               FOR #li_Counter_Hor := 1 TO 3 DO
                   FOR #li_Counter_Ver := 1 TO 3 DO
                       IF ("gtyp_VGR".s_HBW_Outsource_Typ = "gtyp_HBW".Rack_Workpiece[#li_Counter_Ver, #li_Counter_Hor].s_type)
                           AND (#lldt_Outsource > "gtyp_HBW".Rack_History[#li_Counter_Ver, #li_Counter_Hor].History[3].ldt_ts)
                           AND NOT ("gtyp_HBW".Rack_History[#li_Counter_Ver, #li_Counter_Hor].History[3].ldt_ts = LDT#1970-01-01-00:00:00) THEN
                           #lldt_Outsource := "gtyp_HBW".Rack_History[#li_Counter_Ver, #li_Counter_Hor].History[3].ldt_ts;
                           #li_Counter_Act_Hor := #li_Counter_Hor;
                           #li_Counter_Act_Ver := #li_Counter_Ver;
                           #ldi_PosRack_Horizontal := "gtyp_HBW".Rack_Pos[#li_Counter_Ver, #li_Counter_Hor].di_PosRack_Horizontal;
                           #ldi_PosRack_Vertical := "gtyp_HBW".Rack_Pos[#li_Counter_Ver, #li_Counter_Hor].di_PosRack_Vertical;
                       END_IF;
                   END_FOR;
               END_FOR;

               IF (#li_Counter_Act_Hor = 4) OR (#li_Counter_Act_Ver = 4) THEN
                   #li_StepCase := 40;
               ELSE
                   #li_StepCase := 70;
               END_IF;

           70: // Position vertical/horizontal HBW
               "gtyp_HBW".Horizontal_Axis.di_Target_Position := #ldi_PosRack_Horizontal;
               "gtyp_HBW".Horizontal_Axis.x_Start_Positioning := TRUE;
               "gtyp_HBW".Vertical_Axis.di_Target_Position := #ldi_PosRack_Vertical;
               "gtyp_HBW".Vertical_Axis.x_Start_Positioning := TRUE;

               IF ("gtyp_HBW".Horizontal_Axis.di_Actual_Position <= (#ldi_PosRack_Horizontal + "gtyp_HBW".Horizontal_Axis.Config.di_Pos_Window))
                   AND ("gtyp_HBW".Horizontal_Axis.di_Actual_Position >= (#ldi_PosRack_Horizontal - "gtyp_HBW".Horizontal_Axis.Config.di_Pos_Window))
                   AND "gtyp_HBW".Horizontal_Axis.x_Position_Reached THEN
                   "gtyp_HBW".Horizontal_Axis.x_Start_Positioning := FALSE;
               END_IF;

               IF ("gtyp_HBW".Vertical_Axis.di_Actual_Position <= (#ldi_PosRack_Vertical + "gtyp_HBW".Vertical_Axis.Config.di_Pos_Window))
                   AND ("gtyp_HBW".Vertical_Axis.di_Actual_Position >= (#ldi_PosRack_Vertical - "gtyp_HBW".Vertical_Axis.Config.di_Pos_Window))
                   AND "gtyp_HBW".Vertical_Axis.x_Position_Reached THEN
                   "gtyp_HBW".Vertical_Axis.x_Start_Positioning := FALSE;
               END_IF;

               IF ("gtyp_HBW".Horizontal_Axis.di_Actual_Position <= (#ldi_PosRack_Horizontal + "gtyp_HBW".Horizontal_Axis.Config.di_Pos_Window))
                   AND ("gtyp_HBW".Horizontal_Axis.di_Actual_Position >= (#ldi_PosRack_Horizontal - "gtyp_HBW".Horizontal_Axis.Config.di_Pos_Window))
                   AND "gtyp_HBW".Horizontal_Axis.x_Position_Reached
                   AND ("gtyp_HBW".Vertical_Axis.di_Actual_Position <= (#ldi_PosRack_Vertical + "gtyp_HBW".Vertical_Axis.Config.di_Pos_Window))
                   AND ("gtyp_HBW".Vertical_Axis.di_Actual_Position >= (#ldi_PosRack_Vertical - "gtyp_HBW".Vertical_Axis.Config.di_Pos_Window))
                   AND "gtyp_HBW".Vertical_Axis.x_Position_Reached THEN
                   "gtyp_HBW".Horizontal_Axis.x_Start_Positioning := FALSE;
                   "gtyp_HBW".Vertical_Axis.x_Start_Positioning := FALSE;
                   #li_StepCase := 80;
               END_IF;

           80: // Position Cantilever Forward HBW

               "QX_HBW_M4_CantileverBackward_Q8" := FALSE;
               "QX_HBW_M4_CantileverForward_Q7" := TRUE;

               IF "IX_HBW_SwitchCantileverFront_I5" AND NOT "IX_HBW_SwitchCantileverBack_I6" THEN
                   "QX_HBW_M4_CantileverBackward_Q8" := FALSE;
                   "QX_HBW_M4_CantileverForward_Q7" := FALSE;
                   #li_StepCase := 90;
               END_IF;

           90: // Position vertical+offset HBW
               "gtyp_HBW".Vertical_Axis.di_Target_Position := #ldi_PosRack_Vertical - "gtyp_HBW".di_Offset_Pos_Rack_Vertical;
               "gtyp_HBW".Vertical_Axis.x_Start_Positioning := TRUE;

               IF ("gtyp_HBW".Vertical_Axis.di_Actual_Position <= (#ldi_PosRack_Vertical - "gtyp_HBW".di_Offset_Pos_Rack_Vertical + "gtyp_HBW".Vertical_Axis.Config.di_Pos_Window))
                   AND ("gtyp_HBW".Vertical_Axis.di_Actual_Position >= (#ldi_PosRack_Vertical - "gtyp_HBW".di_Offset_Pos_Rack_Vertical - "gtyp_HBW".Vertical_Axis.Config.di_Pos_Window))
                   AND "gtyp_HBW".Vertical_Axis.x_Position_Reached THEN
                   "gtyp_HBW".Vertical_Axis.x_Start_Positioning := FALSE;
                   #li_StepCase := 100;
               END_IF;

           100: // Position vertical Back HBW

               "QX_HBW_M4_CantileverBackward_Q8" := TRUE;
               "QX_HBW_M4_CantileverForward_Q7" := FALSE;

               IF NOT "IX_HBW_SwitchCantileverFront_I5" AND "IX_HBW_SwitchCantileverBack_I6" THEN
                   IF "gtyp_VGR".x_HBW_Storage THEN
                       "gtyp_HBW".Rack_Workpiece[#li_Counter_Act_Ver, #li_Counter_Act_Hor].s_id := '';
                   ELSIF "gtyp_VGR".x_HBW_Outsource THEN
                       "gtyp_Interface_Dashboard".Subscribe.State_HBW.x_active := TRUE;
                       "gtyp_HBW".History := "gtyp_HBW".Rack_History[#li_Counter_Act_Ver, #li_Counter_Act_Hor].History;
                       "gtyp_HBW".Workpiece := "gtyp_HBW".Rack_Workpiece[#li_Counter_Act_Ver, #li_Counter_Act_Hor];
                       #li_Return_LDT := RD_SYS_T(#ldt_MQTT);
                       "gtyp_HBW".History[4].i_code := 400;
                       "gtyp_HBW".History[4].ldt_ts := DT_TO_LDT(#ldt_MQTT);

                       "gtyp_HBW".Rack_Workpiece[#li_Counter_Act_Ver, #li_Counter_Act_Hor].s_id := '';
                       "gtyp_HBW".Rack_Workpiece[#li_Counter_Act_Ver, #li_Counter_Act_Hor].s_state := '';
                       "gtyp_HBW".Rack_Workpiece[#li_Counter_Act_Ver, #li_Counter_Act_Hor].s_type := '';
                       FOR #li_Counter := 1 TO 8 DO
                           "gtyp_HBW".Rack_History[#li_Counter_Act_Ver, #li_Counter_Act_Hor].History[#li_Counter].i_code := 0;
                           "gtyp_HBW".Rack_History[#li_Counter_Act_Ver, #li_Counter_Act_Hor].History[#li_Counter].ldt_ts := DT#1990-01-01-00:00:00;
                       END_FOR;
                   END_IF;
                   "QX_HBW_M4_CantileverBackward_Q8" := FALSE;
                   "QX_HBW_M4_CantileverForward_Q7" := FALSE;
                   #li_StepCase := 110;
               END_IF;

           110: // homing vertical/horizontal axis

               "gtyp_HBW".Horizontal_Axis.x_Reference := TRUE;

               "gtyp_HBW".Vertical_Axis.di_Target_Position := "gtyp_HBW".di_PosBelt_Vertical - "gtyp_HBW".di_Offset_Pos_Belt_Vertical;
               "gtyp_HBW".Vertical_Axis.x_Start_Positioning := TRUE;

               IF ("gtyp_HBW".Vertical_Axis.di_Actual_Position <= ("gtyp_HBW".di_PosBelt_Vertical - "gtyp_HBW".di_Offset_Pos_Belt_Vertical + "gtyp_HBW".Vertical_Axis.Config.di_Pos_Window))
                   AND ("gtyp_HBW".Vertical_Axis.di_Actual_Position >= ("gtyp_HBW".di_PosBelt_Vertical - "gtyp_HBW".di_Offset_Pos_Belt_Vertical - "gtyp_HBW".Vertical_Axis.Config.di_Pos_Window))
                   AND "gtyp_HBW".Vertical_Axis.x_Position_Reached THEN
                   "gtyp_HBW".Vertical_Axis.x_Start_Positioning := FALSE;
               END_IF;

               IF NOT "gtyp_HBW".Horizontal_Axis.x_Referenced THEN
                   #li_StepCase := 120;
               END_IF;

           120: //homed vertical/horizontal axis

               IF "gtyp_HBW".Horizontal_Axis.x_Referenced THEN
                   "gtyp_HBW".Horizontal_Axis.x_Reference := FALSE;
               END_IF;

               IF ("gtyp_HBW".Vertical_Axis.di_Actual_Position <= ("gtyp_HBW".di_PosBelt_Vertical - "gtyp_HBW".di_Offset_Pos_Belt_Vertical + "gtyp_HBW".Vertical_Axis.Config.di_Pos_Window))
                   AND ("gtyp_HBW".Vertical_Axis.di_Actual_Position >= ("gtyp_HBW".di_PosBelt_Vertical - "gtyp_HBW".di_Offset_Pos_Belt_Vertical - "gtyp_HBW".Vertical_Axis.Config.di_Pos_Window))
                   AND "gtyp_HBW".Vertical_Axis.x_Position_Reached THEN
                   "gtyp_HBW".Vertical_Axis.x_Start_Positioning := FALSE;
               END_IF;

               IF "gtyp_HBW".Horizontal_Axis.x_Referenced
                   AND ("gtyp_HBW".Vertical_Axis.di_Actual_Position <= ("gtyp_HBW".di_PosBelt_Vertical - "gtyp_HBW".di_Offset_Pos_Belt_Vertical + "gtyp_HBW".Vertical_Axis.Config.di_Pos_Window))
                   AND ("gtyp_HBW".Vertical_Axis.di_Actual_Position >= ("gtyp_HBW".di_PosBelt_Vertical - "gtyp_HBW".di_Offset_Pos_Belt_Vertical - "gtyp_HBW".Vertical_Axis.Config.di_Pos_Window))
                   AND "gtyp_HBW".Vertical_Axis.x_Position_Reached THEN
                   "gtyp_HBW".Horizontal_Axis.x_Reference := FALSE;
                   "gtyp_HBW".Vertical_Axis.x_Start_Positioning := FALSE;
                   #li_StepCase := 130;
               END_IF;

           130: // Position vertical+offset/horizontal Belt
               "gtyp_HBW".Horizontal_Axis.di_Target_Position := "gtyp_HBW".di_PosBelt_Horizontal;
               "gtyp_HBW".Horizontal_Axis.x_Start_Positioning := TRUE;

               IF ("gtyp_HBW".Horizontal_Axis.di_Actual_Position <= ("gtyp_HBW".di_PosBelt_Horizontal + "gtyp_HBW".Horizontal_Axis.Config.di_Pos_Window))
                   AND ("gtyp_HBW".Horizontal_Axis.di_Actual_Position >= ("gtyp_HBW".di_PosBelt_Horizontal - "gtyp_HBW".Horizontal_Axis.Config.di_Pos_Window))
                   AND "gtyp_HBW".Horizontal_Axis.x_Position_Reached THEN
                   "gtyp_HBW".Horizontal_Axis.x_Start_Positioning := FALSE;
               END_IF;

               IF ("gtyp_HBW".Horizontal_Axis.di_Actual_Position <= ("gtyp_HBW".di_PosBelt_Horizontal + "gtyp_HBW".Horizontal_Axis.Config.di_Pos_Window))
                   AND ("gtyp_HBW".Horizontal_Axis.di_Actual_Position >= ("gtyp_HBW".di_PosBelt_Horizontal - "gtyp_HBW".Horizontal_Axis.Config.di_Pos_Window))
                   AND "gtyp_HBW".Horizontal_Axis.x_Position_Reached THEN
                   "gtyp_HBW".Horizontal_Axis.x_Start_Positioning := FALSE;
                   #li_StepCase := 140;
               END_IF;

           140: // Position cantilever Forward Belt

               "QX_HBW_M4_CantileverBackward_Q8" := FALSE;
               "QX_HBW_M4_CantileverForward_Q7" := TRUE;

               #lx_Time_Error := TRUE;

               IF "IX_HBW_SwitchCantileverFront_I5" AND NOT "IX_HBW_SwitchCantileverBack_I6" THEN
                   "QX_HBW_M4_CantileverBackward_Q8" := FALSE;
                   "QX_HBW_M4_CantileverForward_Q7" := FALSE;
                   #lx_Time_Error := FALSE;
                   #li_StepCase := 150;
               END_IF;

               // runtime error
               IF #lfb_TON_Error.Q THEN
                   #li_Lights := 4;
                   #lx_Time_Error := FALSE;
                   "QX_HBW_M1_ConveyorBeltBackward_Q2" := FALSE;
                   "QX_HBW_M1_ConveyorBeltForward_Q1" := FALSE;
                   "gtyp_Interface_Dashboard".Subscribe.State_HBW.x_active := FALSE;
                   "gtyp_HBW".x_Error := TRUE;
                   #li_StepCase := 0;
               END_IF;

           150: // Position vertical Belt
               "gtyp_HBW".Vertical_Axis.di_Target_Position := "gtyp_HBW".di_PosBelt_Vertical;
               "gtyp_HBW".Vertical_Axis.x_Start_Positioning := TRUE;

               IF ("gtyp_HBW".Vertical_Axis.di_Actual_Position <= ("gtyp_HBW".di_PosBelt_Vertical + "gtyp_HBW".Vertical_Axis.Config.di_Pos_Window))
                   AND ("gtyp_HBW".Vertical_Axis.di_Actual_Position >= ("gtyp_HBW".di_PosBelt_Vertical - "gtyp_HBW".Vertical_Axis.Config.di_Pos_Window))
                   AND "gtyp_HBW".Vertical_Axis.x_Position_Reached THEN
                   "gtyp_HBW".Vertical_Axis.x_Start_Positioning := FALSE;
                   #li_StepCase := 160;
               END_IF;

           160: // Start Conveyor Belt Forward

               #lx_Time_Error := TRUE;

               IF NOT "IX_HBW_LightBarrierInside_I2" THEN
                   "QX_HBW_M1_ConveyorBeltBackward_Q2" := FALSE;
                   "QX_HBW_M1_ConveyorBeltForward_Q1" := TRUE;
                   #lx_Time_Error := FALSE;
                   #li_StepCase := 170;
               END_IF;

               // runtime error
               IF #lfb_TON_Error.Q THEN
                   #li_Lights := 4;
                   #lx_Time_Error := FALSE;
                   "QX_HBW_M1_ConveyorBeltBackward_Q2" := FALSE;
                   "QX_HBW_M1_ConveyorBeltForward_Q1" := FALSE;
                   "gtyp_Interface_Dashboard".Subscribe.State_HBW.x_active := FALSE;
                   "gtyp_HBW".x_Error := TRUE;
                   #li_StepCase := 0;
               END_IF;

           170: //Run-on time reached Conveyor Belt Outside

               #lx_Time_Error := TRUE;

               IF #lfb_TON_ConveyerBelt_Out.Q THEN
                   "QX_HBW_M1_ConveyorBeltBackward_Q2" := FALSE;
                   "QX_HBW_M1_ConveyorBeltForward_Q1" := FALSE;
                   "gtyp_HBW".x_HBW_Container_Available := TRUE;
                   #lx_Time_Error := FALSE;
                   #li_StepCase := 180;
               END_IF;

               // runtime error
               IF #lfb_TON_Error.Q THEN
                   #li_Lights := 4;
                   #lx_Time_Error := FALSE;
                   "QX_HBW_M1_ConveyorBeltBackward_Q2" := FALSE;
                   "QX_HBW_M1_ConveyorBeltForward_Q1" := FALSE;
                   "gtyp_Interface_Dashboard".Subscribe.State_HBW.x_active := FALSE;
                   "gtyp_HBW".x_Error := TRUE;
                   #li_StepCase := 0;
               END_IF;

           180: // VGR picked up - outsource

               #li_Lights := 1;

               IF "gtyp_VGR".x_HBW_PickedUp AND "gtyp_VGR".x_HBW_Outsource THEN
                   "gtyp_VGR".Workpiece := "gtyp_HBW".Workpiece;
                   "gtyp_VGR".History := "gtyp_HBW".History;
                   "gtyp_HBW".Workpiece.s_id := '0';
                   "gtyp_HBW".Workpiece.s_state := '';
                   "gtyp_HBW".Workpiece.s_type := '';
                   FOR #li_Counter := 1 TO 8 DO
                       "gtyp_HBW".History[#li_Counter].i_code := 0;
                       "gtyp_HBW".History[#li_Counter].ldt_ts := DT#1990-01-01-00:00:00;
                   END_FOR;
                   "gtyp_HBW".x_HBW_Container_Available := FALSE;
                   "gtyp_HBW".x_HBW_PickedUp_Accepted := TRUE;

                   "gtyp_Interface_Dashboard".Subscribe.State_HBW.x_active := FALSE;

                   #li_Lights := 2;
                   #li_StepCase := 190;
                   // VGR discard - storage
               ELSIF "gtyp_VGR".x_HBW_Discards AND "gtyp_VGR".x_HBW_Storage THEN
                   "gtyp_Interface_Dashboard".Subscribe.State_HBW.x_active := TRUE;
                   "gtyp_HBW".Workpiece := "gtyp_VGR".Workpiece;
                   "gtyp_HBW".History := "gtyp_VGR".History;
                   "gtyp_HBW".x_HBW_Container_Available := FALSE;
                   "gtyp_HBW".x_HBW_Discards_Accepted := TRUE;
                   #lx_Storage := true;

                   #li_Lights := 2;
                   #li_StepCase := 190;
               END_IF;

           190: // Start Conveyor Belt Back

               IF NOT "gtyp_VGR".x_HBW_Discards AND NOT "gtyp_VGR".x_HBW_PickedUp THEN
                   "QX_HBW_M1_ConveyorBeltBackward_Q2" := TRUE;
                   "QX_HBW_M1_ConveyorBeltForward_Q1" := FALSE;
                   #li_StepCase := 200;
               END_IF;

           200:  // Conveyor Belt inside reached

               #lx_Time_Error := TRUE;

               IF NOT "IX_HBW_LightBarrierInside_I2" THEN
                   "QX_HBW_M1_ConveyorBeltBackward_Q2" := FALSE;
                   "QX_HBW_M1_ConveyorBeltForward_Q1" := FALSE;
                   #lx_Time_Error := FALSE;
                   #li_StepCase := 210;
               END_IF;

               // runtime error
               IF #lfb_TON_Error.Q THEN
                   #li_Lights := 4;
                   #lx_Time_Error := FALSE;
                   "QX_HBW_M1_ConveyorBeltBackward_Q2" := FALSE;
                   "QX_HBW_M1_ConveyorBeltForward_Q1" := FALSE;
                   "gtyp_Interface_Dashboard".Subscribe.State_HBW.x_active := FALSE;
                   "gtyp_HBW".x_Error := TRUE;
                   #li_StepCase := 0;
               END_IF;

           210: // Position vertical+offset Belt

               "gtyp_HBW".Vertical_Axis.di_Target_Position := "gtyp_HBW".di_PosBelt_Vertical - "gtyp_HBW".di_Offset_Pos_Belt_Vertical;
               "gtyp_HBW".Vertical_Axis.x_Start_Positioning := TRUE;

               IF ("gtyp_HBW".Vertical_Axis.di_Actual_Position <= ("gtyp_HBW".di_PosBelt_Vertical - "gtyp_HBW".di_Offset_Pos_Belt_Vertical + "gtyp_HBW".Vertical_Axis.Config.di_Pos_Window))
                   AND ("gtyp_HBW".Vertical_Axis.di_Actual_Position >= ("gtyp_HBW".di_PosBelt_Vertical - "gtyp_HBW".di_Offset_Pos_Belt_Vertical - "gtyp_HBW".Vertical_Axis.Config.di_Pos_Window))
                   AND "gtyp_HBW".Vertical_Axis.x_Position_Reached THEN
                   "gtyp_HBW".Vertical_Axis.x_Start_Positioning := FALSE;
               END_IF;

               IF ("gtyp_HBW".Vertical_Axis.di_Actual_Position <= ("gtyp_HBW".di_PosBelt_Vertical - "gtyp_HBW".di_Offset_Pos_Belt_Vertical + "gtyp_HBW".Vertical_Axis.Config.di_Pos_Window))
                   AND ("gtyp_HBW".Vertical_Axis.di_Actual_Position >= ("gtyp_HBW".di_PosBelt_Vertical - "gtyp_HBW".di_Offset_Pos_Belt_Vertical - "gtyp_HBW".Vertical_Axis.Config.di_Pos_Window))
                   AND "gtyp_HBW".Vertical_Axis.x_Position_Reached THEN
                   "gtyp_HBW".Vertical_Axis.x_Start_Positioning := FALSE;
                   #li_StepCase := 220;
               END_IF;

           220: // Position Cantilever back Belt   
               "QX_HBW_M4_CantileverBackward_Q8" := TRUE;
               "QX_HBW_M4_CantileverForward_Q7" := FALSE;

               IF NOT "IX_HBW_SwitchCantileverFront_I5" AND "IX_HBW_SwitchCantileverBack_I6" THEN
                   "QX_HBW_M4_CantileverBackward_Q8" := FALSE;
                   "QX_HBW_M4_CantileverForward_Q7" := FALSE;
                   #li_StepCase := 230;
               END_IF;

           230: // Position vertical+offset/horizontal HBW
               "gtyp_HBW".Horizontal_Axis.di_Target_Position := #ldi_PosRack_Horizontal;
               "gtyp_HBW".Horizontal_Axis.x_Start_Positioning := TRUE;
               "gtyp_HBW".Vertical_Axis.di_Target_Position := #ldi_PosRack_Vertical - "gtyp_HBW".di_Offset_Pos_Rack_Vertical;
               "gtyp_HBW".Vertical_Axis.x_Start_Positioning := TRUE;

               IF ("gtyp_HBW".Horizontal_Axis.di_Actual_Position <= (#ldi_PosRack_Horizontal + "gtyp_HBW".Horizontal_Axis.Config.di_Pos_Window))
                   AND ("gtyp_HBW".Horizontal_Axis.di_Actual_Position >= (#ldi_PosRack_Horizontal - "gtyp_HBW".Horizontal_Axis.Config.di_Pos_Window))
                   AND "gtyp_HBW".Horizontal_Axis.x_Position_Reached THEN
                   "gtyp_HBW".Horizontal_Axis.x_Start_Positioning := FALSE;
               END_IF;

               IF ("gtyp_HBW".Vertical_Axis.di_Actual_Position <= (#ldi_PosRack_Vertical - "gtyp_HBW".di_Offset_Pos_Rack_Vertical + "gtyp_HBW".Vertical_Axis.Config.di_Pos_Window))
                   AND ("gtyp_HBW".Vertical_Axis.di_Actual_Position >= (#ldi_PosRack_Vertical - "gtyp_HBW".di_Offset_Pos_Rack_Vertical - "gtyp_HBW".Vertical_Axis.Config.di_Pos_Window))
                   AND "gtyp_HBW".Vertical_Axis.x_Position_Reached THEN
                   "gtyp_HBW".Vertical_Axis.x_Start_Positioning := FALSE;
               END_IF;

               IF ("gtyp_HBW".Horizontal_Axis.di_Actual_Position <= (#ldi_PosRack_Horizontal + "gtyp_HBW".Horizontal_Axis.Config.di_Pos_Window))
                   AND ("gtyp_HBW".Horizontal_Axis.di_Actual_Position >= (#ldi_PosRack_Horizontal - "gtyp_HBW".Horizontal_Axis.Config.di_Pos_Window))
                   AND "gtyp_HBW".Horizontal_Axis.x_Position_Reached
                   AND ("gtyp_HBW".Vertical_Axis.di_Actual_Position <= (#ldi_PosRack_Vertical - "gtyp_HBW".di_Offset_Pos_Rack_Vertical + "gtyp_HBW".Vertical_Axis.Config.di_Pos_Window))
                   AND ("gtyp_HBW".Vertical_Axis.di_Actual_Position >= (#ldi_PosRack_Vertical - "gtyp_HBW".di_Offset_Pos_Rack_Vertical - "gtyp_HBW".Vertical_Axis.Config.di_Pos_Window))
                   AND "gtyp_HBW".Vertical_Axis.x_Position_Reached THEN
                   "gtyp_HBW".Horizontal_Axis.x_Start_Positioning := FALSE;
                   "gtyp_HBW".Vertical_Axis.x_Start_Positioning := FALSE;
                   #li_StepCase := 240;
               END_IF;

           240: // Position Cantilever Forward HBW

               "QX_HBW_M4_CantileverBackward_Q8" := FALSE;
               "QX_HBW_M4_CantileverForward_Q7" := TRUE;

               IF "IX_HBW_SwitchCantileverFront_I5" AND NOT "IX_HBW_SwitchCantileverBack_I6" THEN
                   "QX_HBW_M4_CantileverBackward_Q8" := FALSE;
                   "QX_HBW_M4_CantileverForward_Q7" := FALSE;
                   #li_StepCase := 250;
               END_IF;

           250: // Position vertical HBW
               "gtyp_HBW".Vertical_Axis.di_Target_Position := #ldi_PosRack_Vertical;
               "gtyp_HBW".Vertical_Axis.x_Start_Positioning := TRUE;

               IF ("gtyp_HBW".Vertical_Axis.di_Actual_Position <= (#ldi_PosRack_Vertical + "gtyp_HBW".Vertical_Axis.Config.di_Pos_Window))
                   AND ("gtyp_HBW".Vertical_Axis.di_Actual_Position >= (#ldi_PosRack_Vertical - "gtyp_HBW".Vertical_Axis.Config.di_Pos_Window))
                   AND "gtyp_HBW".Vertical_Axis.x_Position_Reached THEN
                   IF #lx_Storage THEN
                       #li_Return_LDT := RD_SYS_T(#ldt_MQTT);
                       "gtyp_HBW".History[3].i_code := 300;
                       "gtyp_HBW".History[3].ldt_ts := DT_TO_LDT(#ldt_MQTT);
                       "gtyp_HBW".Rack_Workpiece[#li_Counter_Act_Ver, #li_Counter_Act_Hor] := "gtyp_HBW".Workpiece;
                       "gtyp_HBW".Rack_History[#li_Counter_Act_Ver, #li_Counter_Act_Hor].History := "gtyp_HBW".History;
                       "gtyp_Interface_Dashboard".Subscribe.State_HBW.x_active := FALSE;
                   ELSE
                       "gtyp_HBW".Rack_Workpiece[#li_Counter_Act_Ver, #li_Counter_Act_Hor].s_id := '0';
                   END_IF;
                   "gtyp_HBW".Vertical_Axis.x_Start_Positioning := FALSE;
                   #li_StepCase := 260;
               END_IF;

           260: // Position Cantilever Backward HBW

               "QX_HBW_M4_CantileverBackward_Q8" := TRUE;
               "QX_HBW_M4_CantileverForward_Q7" := FALSE;

               IF NOT "IX_HBW_SwitchCantileverFront_I5" AND "IX_HBW_SwitchCantileverBack_I6" THEN
                   "QX_HBW_M4_CantileverBackward_Q8" := FALSE;
                   "QX_HBW_M4_CantileverForward_Q7" := FALSE;
                   #li_StepCase := 0;
                   #lx_Storage := FALSE;
               END_IF;
               // Statement section ELSE    
           ELSE
               ;
       END_CASE;

       //Reset the information in the high-bay warehouse
       IF "gtyp_Setup".x_Clean_Rack_HBW THEN
           FOR #li_Counter_Hor := 1 TO 3 DO
               FOR #li_Counter_Ver := 1 TO 3 DO
                   "gtyp_HBW".Rack_Workpiece[#li_Counter_Ver, #li_Counter_Hor].s_id := '0';
                   "gtyp_HBW".Rack_Workpiece[#li_Counter_Ver, #li_Counter_Hor].s_state := '';
                   "gtyp_HBW".Rack_Workpiece[#li_Counter_Ver, #li_Counter_Hor].s_type := '';
                   FOR #li_Counter := 1 TO 8 DO
                       "gtyp_HBW".Rack_History[#li_Counter_Ver, #li_Counter_Hor].History[#li_Counter].i_code := 0;
                       "gtyp_HBW".Rack_History[#li_Counter_Ver, #li_Counter_Hor].History[#li_Counter].ldt_ts := DT#1990-01-01-00:00:00;
                   END_FOR;
               END_FOR;
           END_FOR;
           "gtyp_Setup".x_Clean_Rack_HBW := FALSE;
       END_IF;

       // reload PWM
       "QW_HBW_PWM_ConveyorBelt_M1" := "gtyp_HBW"."i_PWM_ConveyorBelt";
       "QW_HBW_PWM_Cantilever_M4" := "gtyp_HBW"."i_PWM_Cantilever";
   ELSE
       FOR #li_Counter_Hor := 1 TO 3 DO
           FOR #li_Counter_Ver := 1 TO 3 DO
               IF "gtyp_HBW".Rack_Workpiece[#li_Counter_Ver, #li_Counter_Hor].s_id = '' THEN
                   "gtyp_HBW".Rack_Workpiece[#li_Counter_Ver, #li_Counter_Hor].s_id := '0';
                   "gtyp_HBW".Rack_Workpiece[#li_Counter_Ver, #li_Counter_Hor].s_state := '';
                   "gtyp_HBW".Rack_Workpiece[#li_Counter_Ver, #li_Counter_Hor].s_type := '';
                   FOR #li_Counter := 1 TO 8 DO
                       "gtyp_HBW".Rack_History[#li_Counter_Ver, #li_Counter_Hor].History[#li_Counter].i_code := 0;
                       "gtyp_HBW".Rack_History[#li_Counter_Ver, #li_Counter_Hor].History[#li_Counter].ldt_ts := DT#1990-01-01-00:00:00;
                   END_FOR;
               END_IF;
           END_FOR;
       END_FOR;

       "gtyp_HBW".x_Start_Park_Position := FALSE;
       "gtyp_HBW".x_Park_Position_Reached := FALSE;
       "gtyp_HBW".x_HBW_PickedUp_Accepted := FALSE;
       "gtyp_HBW".x_HBW_Discards_Accepted := FALSE;
       "gtyp_HBW".x_HBW_PickUp_Ready := FALSE;
       "gtyp_HBW".x_HBW_Container_Available := FALSE;
       "gtyp_HBW".x_Error := FALSE;

       #li_Lights := 1;
       #lx_Start_TON_Fill_HBW := TRUE;
       #lx_Init := TRUE;
   END_IF;
END_FUNCTION_BLOCK

FUNCTION_BLOCK "PRG_HBW_Axis_Horizontal_Act_Pos"   // FB26, SCL
TITLE = Program Axis horizontal Actual Position
{ S7_Optimized_Access := 'TRUE' }
AUTHOR : A.Schaefer
VERSION : 0.0
   VAR
      lfb_IN_DEC : "FB_INC_DEC";
   END_VAR
BEGIN
   // FB increment axis
   #lfb_IN_DEC(inx_CHa := "IX_HBW_EncoderHorizontalAxisImp2_B2",
               inx_CHb := "IX_HBW_EncoderHorizontalAxisImp1_B1",
               ini_Ref_Wert := DINT_TO_INT("gtyp_HBW".Horizontal_Axis.Config.di_Ref_Pos),
               inx_RST := "IX_HBW_RefSwitchHorizontalAxis_I1");

   "gtyp_HBW".Horizontal_Axis.di_Increment := #lfb_IN_DEC.outi_cnt;
END_FUNCTION_BLOCK

FUNCTION_BLOCK "PRG_HBW_Axis_Vertical_Act_Pos"   // FB27, SCL
TITLE = Program Axis vertical Actual Position
{ S7_Optimized_Access := 'TRUE' }
AUTHOR : A.Schaefer
VERSION : 0.0
   VAR
      lfb_IN_DEC : "FB_INC_DEC";
   END_VAR
BEGIN
   // FB increment axis
   #lfb_IN_DEC(inx_CHa := "IX_HBW_EncoderVerticalAxisImp1_B3",
               inx_CHb := "IX_HBW_EncoderVerticalAxisImp2_B4",
               ini_Ref_Wert := DINT_TO_INT("gtyp_HBW".Vertical_Axis.Config.di_Ref_Pos),
               inx_RST := "IX_HBW_RefSwitchVerticalAxis_I4");

   "gtyp_HBW".Vertical_Axis.di_Increment := #lfb_IN_DEC.outi_cnt;
END_FUNCTION_BLOCK

FUNCTION_BLOCK "PRG_HBW_Set_Positioning"   // FB31, SCL
TITLE = Program Set Positioning HBW
{ S7_Optimized_Access := 'TRUE' }
AUTHOR : A.Schaefer
VERSION : 0.0
   VAR
      lx_Init : Bool;
      lx_Start_TON_Wait : Bool;
      lx_Start_Positioning_m : Bool;
      lx_Start_FinalPositioning_m : Bool;
      lx_Start_Offset_m : Bool;
      lt_TON_Wait : Time;
      li_Counter_Hor : Int;
      li_Counter_Ver : Int;
      li_Counter_Act_Hor : Int;
      li_Counter_Act_Ver : Int;
      li_Counter : Int;
      li_StepCase : Int;
      ldi_Pos_Horizontal : DInt;
      ldi_Pos_Vertical : DInt;
      ldi_Offset_Vertical : DInt;
      lfb_R_Trig_Deaktivate : R_TRIG;
      lfb_TON_Wait : TON_TIME;
   END_VAR
BEGIN
   IF #lx_Init THEN

       // FB TON Wait
       #lfb_TON_Wait(IN := #lx_Start_TON_Wait,
                     PT := #lt_TON_Wait);

       #lfb_R_Trig_Deaktivate(CLK := NOT "gtyp_Setup".x_Set_Pos_Activ
                              OR NOT (("gtyp_Setup".i_Pos_Selection > 20)
                              AND ("gtyp_Setup".i_Pos_Selection < 41)));
       // Deaktivate step 110   
       IF #lfb_R_Trig_Deaktivate.Q THEN
           "gtyp_HBW".Horizontal_Axis.x_Start_Positioning := FALSE;
           "gtyp_HBW".Vertical_Axis.x_Start_Positioning := FALSE;
           "gtyp_HBW".Horizontal_Axis.x_Reference := FALSE;
           "gtyp_HBW".Vertical_Axis.x_Reference := FALSE;
           "gtyp_Setup".x_Start_Positioning := FALSE;
           "gtyp_Setup".x_Final_Positioning := FALSE;
           "gtyp_Setup".x_Home_Positioning := FALSE;
           "gtyp_Setup".x_Start_Offset := FALSE;
           "QX_HBW_M4_CantileverBackward_Q8" := FALSE;
           "QX_HBW_M4_CantileverForward_Q7" := FALSE;
           IF (#li_StepCase > 10) THEN
               #li_StepCase := 110;
           END_IF;
       END_IF;

       // Set Positioning activ?
       IF "gtyp_Setup".x_Set_Pos_Activ
           AND (("gtyp_Setup".i_Pos_Selection > 20)
           AND ("gtyp_Setup".i_Pos_Selection < 41))
           AND ((#li_StepCase = 40)
           OR (#li_StepCase = 60)
           OR (#li_StepCase = 80)
           OR (#li_StepCase = 100)) THEN

           // Deciding which Position
           // Position - Belt
           IF "gtyp_Setup".i_Pos_Selection = 21 THEN
               #ldi_Pos_Horizontal := "gtyp_HBW".di_PosBelt_Horizontal;
               #ldi_Pos_Vertical := "gtyp_HBW".di_PosBelt_Vertical;
               #ldi_Offset_Vertical := "gtyp_HBW".di_Offset_Pos_Belt_Vertical;
               // Position - A1 
           ELSIF "gtyp_Setup".i_Pos_Selection = 22 THEN
               #ldi_Pos_Horizontal := "gtyp_HBW".di_PosRack_A1_Horizontal;
               #ldi_Pos_Vertical := "gtyp_HBW".di_PosRack_A1_Vertical;
               #ldi_Offset_Vertical := "gtyp_HBW".di_Offset_Pos_Rack_Vertical;
               // Position - B2 
           ELSIF "gtyp_Setup".i_Pos_Selection = 23 THEN
               #ldi_Pos_Horizontal := "gtyp_HBW".di_PosRack_B2_Horizontal;
               #ldi_Pos_Vertical := "gtyp_HBW".di_PosRack_B2_Vertical;
               #ldi_Offset_Vertical := "gtyp_HBW".di_Offset_Pos_Rack_Vertical;
               // Position - C3 
           ELSIF "gtyp_Setup".i_Pos_Selection = 24 THEN
               #ldi_Pos_Horizontal := "gtyp_HBW".di_PosRack_C3_Horizontal;
               #ldi_Pos_Vertical := "gtyp_HBW".di_PosRack_C3_Vertical;
               #ldi_Offset_Vertical := "gtyp_HBW".di_Offset_Pos_Rack_Vertical;
           END_IF;
       END_IF;

       // Set Positioning activ?
       IF NOT "gtyp_Setup".x_Set_Pos_Activ THEN
           "gtyp_Setup".i_Pos_Selection := 0;
       END_IF;

       // step chain HBW
       CASE #li_StepCase OF

           0:  // init
               #lx_Start_TON_Wait := FALSE;
               #li_StepCase := 10;

           10:  // Set Positioning activ?
               IF "gtyp_Setup".x_Set_Pos_Activ
                   AND (("gtyp_Setup".i_Pos_Selection > 20)
                   AND ("gtyp_Setup".i_Pos_Selection < 41)) THEN

                   "gtyp_HBW".Horizontal_Axis.x_Start_Positioning := FALSE;
                   "gtyp_HBW".Vertical_Axis.x_Start_Positioning := FALSE;
                   "gtyp_HBW".Horizontal_Axis.x_Reference := FALSE;
                   "gtyp_HBW".Vertical_Axis.x_Reference := FALSE;
                   "gtyp_Setup".x_Start_Positioning := FALSE;
                   "gtyp_Setup".x_Final_Positioning := FALSE;
                   "gtyp_Setup".x_Home_Positioning := FALSE;
                   "gtyp_Setup".x_Start_Offset := FALSE;
                   "QX_HBW_M4_CantileverBackward_Q8" := FALSE;
                   "QX_HBW_M4_CantileverForward_Q7" := FALSE;
                   #li_StepCase := 20;
               END_IF;

           20: //homing vertical/horizontal axis

               "gtyp_HBW".Horizontal_Axis.x_Reference := TRUE;
               "gtyp_HBW".Vertical_Axis.x_Reference := TRUE;

               IF NOT "gtyp_HBW".Horizontal_Axis.x_Referenced AND NOT "gtyp_HBW".Vertical_Axis.x_Referenced THEN
                   #li_StepCase := 30;
               END_IF;

           30: // homed vertical/horizontal axis
               IF "gtyp_HBW".Horizontal_Axis.x_Referenced THEN
                   "gtyp_HBW".Horizontal_Axis.x_Reference := FALSE;
               END_IF;
               IF "gtyp_HBW".Vertical_Axis.x_Referenced THEN
                   "gtyp_HBW".Vertical_Axis.x_Reference := FALSE;
               END_IF;

               IF "gtyp_HBW".Horizontal_Axis.x_Referenced AND "gtyp_HBW".Vertical_Axis.x_Referenced THEN
                   "gtyp_HBW".Horizontal_Axis.x_Reference := FALSE;
                   "gtyp_HBW".Vertical_Axis.x_Reference := FALSE;
                   #li_StepCase := 40;
               END_IF;

           40: // Start Positioning Step next
               IF "gtyp_Setup".x_Start_Positioning OR #lx_Start_Positioning_m OR #lx_Start_FinalPositioning_m OR #lx_Start_Offset_m THEN
                   #lx_Start_Positioning_m := FALSE;
                   #li_StepCase := 50;
               END_IF;

           50: // Position vertical/horizontal HBW
               "gtyp_HBW".Horizontal_Axis.di_Target_Position := #ldi_Pos_Horizontal;
               "gtyp_HBW".Horizontal_Axis.x_Start_Positioning := TRUE;
               "gtyp_HBW".Vertical_Axis.di_Target_Position := #ldi_Pos_Vertical;
               "gtyp_HBW".Vertical_Axis.x_Start_Positioning := TRUE;

               IF ("gtyp_HBW".Horizontal_Axis.di_Actual_Position <= (#ldi_Pos_Horizontal + "gtyp_HBW".Horizontal_Axis.Config.di_Pos_Window))
                   AND ("gtyp_HBW".Horizontal_Axis.di_Actual_Position >= (#ldi_Pos_Horizontal - "gtyp_HBW".Horizontal_Axis.Config.di_Pos_Window))
                   AND "gtyp_HBW".Horizontal_Axis.x_Position_Reached THEN
                   "gtyp_HBW".Horizontal_Axis.x_Start_Positioning := FALSE;
               END_IF;

               IF ("gtyp_HBW".Vertical_Axis.di_Actual_Position <= (#ldi_Pos_Vertical + "gtyp_HBW".Vertical_Axis.Config.di_Pos_Window))
                   AND ("gtyp_HBW".Vertical_Axis.di_Actual_Position >= (#ldi_Pos_Vertical - "gtyp_HBW".Vertical_Axis.Config.di_Pos_Window))
                   AND "gtyp_HBW".Vertical_Axis.x_Position_Reached THEN
                   "gtyp_HBW".Vertical_Axis.x_Start_Positioning := FALSE;
               END_IF;

               IF ("gtyp_HBW".Horizontal_Axis.di_Actual_Position <= (#ldi_Pos_Horizontal + "gtyp_HBW".Horizontal_Axis.Config.di_Pos_Window))
                   AND ("gtyp_HBW".Horizontal_Axis.di_Actual_Position >= (#ldi_Pos_Horizontal - "gtyp_HBW".Horizontal_Axis.Config.di_Pos_Window))
                   AND "gtyp_HBW".Horizontal_Axis.x_Position_Reached
                   AND ("gtyp_HBW".Vertical_Axis.di_Actual_Position <= (#ldi_Pos_Vertical + "gtyp_HBW".Vertical_Axis.Config.di_Pos_Window))
                   AND ("gtyp_HBW".Vertical_Axis.di_Actual_Position >= (#ldi_Pos_Vertical - "gtyp_HBW".Vertical_Axis.Config.di_Pos_Window))
                   AND "gtyp_HBW".Vertical_Axis.x_Position_Reached THEN
                   "gtyp_HBW".Horizontal_Axis.x_Start_Positioning := FALSE;
                   "gtyp_HBW".Vertical_Axis.x_Start_Positioning := FALSE;
                   "gtyp_Setup".x_Start_Positioning := FALSE;
                   #li_StepCase := 60;
               END_IF;

           60: // Deciding which doing

               // Start new Positioning
               IF "gtyp_Setup".x_Start_Positioning THEN
                   #lx_Start_Positioning_m := TRUE;
                   #li_StepCase := 10;
                   // Start Final Positioning
               ELSIF "gtyp_Setup".x_Final_Positioning OR #lx_Start_FinalPositioning_m OR #lx_Start_Offset_m THEN
                   #lx_Start_FinalPositioning_m := FALSE;
                   #li_StepCase := 70;
                   // Deaktivate Set Positioning
               ELSIF #lfb_R_Trig_Deaktivate.Q OR "gtyp_Setup".x_Home_Positioning THEN
                   "gtyp_Setup".x_Home_Positioning := FALSE;
                   #li_StepCase := 110;
               END_IF;

           70: // Final Positioning - Cantilever Forward

               "QX_HBW_M4_CantileverBackward_Q8" := FALSE;
               "QX_HBW_M4_CantileverForward_Q7" := TRUE;

               IF "IX_HBW_SwitchCantileverFront_I5" AND NOT "IX_HBW_SwitchCantileverBack_I6" THEN
                   "QX_HBW_M4_CantileverBackward_Q8" := FALSE;
                   "QX_HBW_M4_CantileverForward_Q7" := FALSE;
                   "gtyp_Setup".x_Final_Positioning := FALSE;
                   #li_StepCase := 80;
               END_IF;

           80: // Deciding which doing

               // Start new Positioning
               IF "gtyp_Setup".x_Start_Positioning THEN
                   #lx_Start_Positioning_m := TRUE;
                   #li_StepCase := 110;
                   // Start Final Positioning
               ELSIF "gtyp_Setup".x_Final_Positioning THEN
                   #lx_Start_FinalPositioning_m := TRUE;
                   #li_StepCase := 110;
                   // Start Final Positioning
               ELSIF "gtyp_Setup".x_Start_Offset OR #lx_Start_Offset_m THEN
                   #lx_Start_Offset_m := FALSE;
                   #li_StepCase := 90;
                   // Deaktivate Set Positioning
               ELSIF #lfb_R_Trig_Deaktivate.Q OR "gtyp_Setup".x_Home_Positioning THEN
                   "gtyp_Setup".x_Home_Positioning := FALSE;
                   #li_StepCase := 110;
               END_IF;

           90: // Position vertical+offset HBW
               "gtyp_HBW".Vertical_Axis.di_Target_Position := #ldi_Pos_Vertical - #ldi_Offset_Vertical;
               "gtyp_HBW".Vertical_Axis.x_Start_Positioning := TRUE;

               IF ("gtyp_HBW".Vertical_Axis.di_Actual_Position <= (#ldi_Pos_Vertical - #ldi_Offset_Vertical + "gtyp_HBW".Vertical_Axis.Config.di_Pos_Window))
                   AND ("gtyp_HBW".Vertical_Axis.di_Actual_Position >= (#ldi_Pos_Vertical - #ldi_Offset_Vertical - "gtyp_HBW".Vertical_Axis.Config.di_Pos_Window))
                   AND "gtyp_HBW".Vertical_Axis.x_Position_Reached THEN
                   "gtyp_HBW".Vertical_Axis.x_Start_Positioning := FALSE;
                   "gtyp_Setup".x_Start_Offset := FALSE;
                   #li_StepCase := 100;
               END_IF;

           100: // Deciding which doing

               // Start new Positioning
               IF "gtyp_Setup".x_Start_Positioning THEN
                   #lx_Start_Positioning_m := TRUE;
                   #li_StepCase := 110;
                   // Start Final Positioning
               ELSIF "gtyp_Setup".x_Final_Positioning THEN
                   #lx_Start_FinalPositioning_m := TRUE;
                   #li_StepCase := 110;
                   // Start Final Positioning
               ELSIF "gtyp_Setup".x_Start_Offset THEN
                   #lx_Start_Offset_m := true;
                   #li_StepCase := 110;
                   // Deaktivate Set Positioning
               ELSIF #lfb_R_Trig_Deaktivate.Q OR "gtyp_Setup".x_Home_Positioning THEN
                   "gtyp_Setup".x_Home_Positioning := FALSE;
                   #li_StepCase := 110;
               END_IF;

           110: // Position vertical HBW
               "gtyp_HBW".Vertical_Axis.di_Target_Position := #ldi_Pos_Vertical;
               "gtyp_HBW".Vertical_Axis.x_Start_Positioning := TRUE;

               IF ("gtyp_HBW".Vertical_Axis.di_Actual_Position <= (#ldi_Pos_Vertical + "gtyp_HBW".Vertical_Axis.Config.di_Pos_Window))
                   AND ("gtyp_HBW".Vertical_Axis.di_Actual_Position >= (#ldi_Pos_Vertical - "gtyp_HBW".Vertical_Axis.Config.di_Pos_Window))
                   AND "gtyp_HBW".Vertical_Axis.x_Position_Reached THEN
                   "gtyp_HBW".Vertical_Axis.x_Start_Positioning := FALSE;
                   #li_StepCase := 120;
               END_IF;

           120: // Position vertical Back HBW

               "QX_HBW_M4_CantileverBackward_Q8" := TRUE;
               "QX_HBW_M4_CantileverForward_Q7" := FALSE;

               IF NOT "IX_HBW_SwitchCantileverFront_I5" AND "IX_HBW_SwitchCantileverBack_I6" THEN
                   "QX_HBW_M4_CantileverBackward_Q8" := FALSE;
                   "QX_HBW_M4_CantileverForward_Q7" := FALSE;
                   #li_StepCase := 130;
               END_IF;

           130: // homing vertical/horizontal axis

               "gtyp_HBW".Horizontal_Axis.x_Reference := TRUE;
               "gtyp_HBW".Vertical_Axis.x_Reference := TRUE;

               IF NOT "gtyp_HBW".Horizontal_Axis.x_Referenced AND NOT "gtyp_HBW".Vertical_Axis.x_Referenced THEN
                   #li_StepCase := 140;
               END_IF;

           140: //homed vertical/horizontal axis
               IF "gtyp_HBW".Horizontal_Axis.x_Referenced THEN
                   "gtyp_HBW".Horizontal_Axis.x_Reference := FALSE;
               END_IF;
               IF "gtyp_HBW".Vertical_Axis.x_Referenced THEN
                   "gtyp_HBW".Vertical_Axis.x_Reference := FALSE;
               END_IF;

               IF "gtyp_HBW".Horizontal_Axis.x_Referenced AND "gtyp_HBW".Vertical_Axis.x_Referenced THEN
                   "gtyp_HBW".Horizontal_Axis.x_Reference := FALSE;
                   "gtyp_HBW".Vertical_Axis.x_Reference := FALSE;
                   #li_StepCase := 0;
               END_IF;

               // Statement section ELSE    
           ELSE
               ;
       END_CASE;

       IF (("gtyp_Setup".i_Pos_Selection > 20)
           AND ("gtyp_Setup".i_Pos_Selection < 41)) THEN
           // Reload Pos Value
           "gtyp_Setup".di_Pos_Horizontal := #ldi_Pos_Horizontal;
           "gtyp_Setup".di_Pos_Vertical := #ldi_Pos_Vertical;
           "gtyp_Setup".di_Pos_Rotate := 0;
       END_IF;
   ELSE
       #lx_Init := TRUE;
   END_IF;
END_FUNCTION_BLOCK

FUNCTION_BLOCK "PRG_HBW_Set_Park_Position"   // FB40, SCL
TITLE = Program Set Positioning HBW
{ S7_Optimized_Access := 'TRUE' }
AUTHOR : A.Schaefer
VERSION : 0.0
   VAR
      lx_Init : Bool;
      lx_Start_TON_Wait : Bool;
      lt_TON_Wait : Time;
      li_StepCase : Int;
      lfb_TON_Wait : TON_TIME;
      lfb_R_Trig_Start_Park_Pos : R_TRIG;
   END_VAR
BEGIN
   IF #lx_Init THEN

       // FB TON Wait
       #lfb_TON_Wait(IN := #lx_Start_TON_Wait,
                     PT := #lt_TON_Wait);

       #lfb_R_Trig_Start_Park_Pos(CLK := "gtyp_Setup".x_Park_Position
                                  OR "IX_Set_Park_Position");

       // Set Start Park Position   
       IF #lfb_R_Trig_Start_Park_Pos.Q THEN
           "gtyp_HBW".x_Start_Park_Position := TRUE;
           #li_StepCase := 0;
       END_IF;

       // not Start Park Pos Step 0
       IF NOT "gtyp_HBW".x_Start_Park_Position THEN
           #li_StepCase := 0;
       END_IF;

       // step chain HBW
       CASE #li_StepCase OF

           0:  // init
               #lx_Start_TON_Wait := FALSE;
               #li_StepCase := 10;

           10:  // Set Positioning activ?
               IF "IX_HBW_SwitchCantileverFront_I5" OR NOT "IX_HBW_SwitchCantileverBack_I6" THEN
                   "QX_HBW_M4_CantileverBackward_Q8" := TRUE;
                   "QX_HBW_M4_CantileverForward_Q7" := FALSE;
               ELSIF NOT "IX_HBW_SwitchCantileverFront_I5" AND "IX_HBW_SwitchCantileverBack_I6" THEN
                   "QX_HBW_M4_CantileverBackward_Q8" := FALSE;
                   "QX_HBW_M4_CantileverForward_Q7" := FALSE;
                   #li_StepCase := 20;
               END_IF;

           20:  // Set Positioning activ?
               IF "gtyp_HBW".x_Start_Park_Position AND NOT "gtyp_HBW".x_Park_Position_Reached THEN
                   "gtyp_HBW".Horizontal_Axis.x_Start_Positioning := FALSE;
                   "gtyp_HBW".Vertical_Axis.x_Start_Positioning := FALSE;
                   "gtyp_HBW".Horizontal_Axis.x_Reference := FALSE;
                   "gtyp_HBW".Vertical_Axis.x_Reference := FALSE;
                   "QX_HBW_M4_CantileverBackward_Q8" := FALSE;
                   "QX_HBW_M4_CantileverForward_Q7" := FALSE;
                   #li_StepCase := 30;
               END_IF;

           30: // homing vertical axis
               "gtyp_HBW".Vertical_Axis.x_Reference := TRUE;

               IF NOT "gtyp_HBW".Vertical_Axis.x_Referenced THEN
                   #li_StepCase := 40;
               END_IF;

           40: // homed vertical axis
               IF "gtyp_HBW".Vertical_Axis.x_Referenced THEN
                   "gtyp_HBW".Vertical_Axis.x_Reference := FALSE;
                   #li_StepCase := 50;
               END_IF;

           50: // homing horizontal axis
               "gtyp_HBW".Horizontal_Axis.x_Reference := TRUE;

               IF NOT "gtyp_HBW".Horizontal_Axis.x_Referenced THEN
                   #li_StepCase := 60;
               END_IF;

           60: // homed horizontal axis
               IF "gtyp_HBW".Horizontal_Axis.x_Referenced THEN
                   "gtyp_HBW".Horizontal_Axis.x_Reference := FALSE;
                   #li_StepCase := 70;
               END_IF;

           70: // Position horizontal Axis
               "gtyp_HBW".Horizontal_Axis.di_Target_Position := "gtyp_HBW".di_Pos_Park_Horizontal;
               "gtyp_HBW".Horizontal_Axis.x_Start_Positioning := TRUE;

               IF ("gtyp_HBW".Horizontal_Axis.di_Actual_Position <= ("gtyp_HBW".di_Pos_Park_Horizontal + "gtyp_HBW".Horizontal_Axis.Config.di_Pos_Window))
                   AND ("gtyp_HBW".Horizontal_Axis.di_Actual_Position >= ("gtyp_HBW".di_Pos_Park_Horizontal - "gtyp_HBW".Horizontal_Axis.Config.di_Pos_Window))
                   AND "gtyp_HBW".Horizontal_Axis.x_Position_Reached THEN
                   "gtyp_HBW".Horizontal_Axis.x_Start_Positioning := FALSE;
                   #li_StepCase := 80;
               END_IF;

           80: // Position vertical Axis
               "gtyp_HBW".Vertical_Axis.di_Target_Position := "gtyp_HBW".di_Pos_Park_Vertical;
               "gtyp_HBW".Vertical_Axis.x_Start_Positioning := TRUE;

               IF ("gtyp_HBW".Vertical_Axis.di_Actual_Position <= ("gtyp_HBW".di_Pos_Park_Vertical + "gtyp_HBW".Vertical_Axis.Config.di_Pos_Window))
                   AND ("gtyp_HBW".Vertical_Axis.di_Actual_Position >= ("gtyp_HBW".di_Pos_Park_Vertical - "gtyp_HBW".Vertical_Axis.Config.di_Pos_Window))
                   AND "gtyp_HBW".Vertical_Axis.x_Position_Reached THEN
                   "gtyp_HBW".Vertical_Axis.x_Start_Positioning := FALSE;
                   #li_StepCase := 90;
               END_IF;

           90: // Deciding which doing
               "gtyp_HBW".x_Park_Position_Reached := TRUE;


               // Statement section ELSE    
           ELSE
               ;
       END_CASE;

   ELSE
       #lx_Init := TRUE;
   END_IF;
END_FUNCTION_BLOCK

// folder: 3.3. MPO

FUNCTION_BLOCK "PRG_MPO_Ablauf"   // FB17, SCL
TITLE = Program Ablauf MPO
{ S7_Optimized_Access := 'TRUE' }
AUTHOR : A.Schaefer
VERSION : 0.0
   VAR
      lx_Init : Bool;
      lx_Start_TON_Wait : Bool;
      lx_Time_Error : Bool;
      lt_TON_Wait : Time;
      lx_Start_TON_State : Bool;
      ldt_MQTT : Date_And_Time;
      li_Return_LDT : Int;
      li_StepCase : Int;
      li_Lights : Int;
      li_Lights_old : Int;
      li_Counter : Int;
      lfb_blinker : "FB_Blinker";
      lfb_TOF_ConveyerBelt_Out : TOF_TIME;
      lfb_TON_Wait : TON_TIME;
      lfb_TON_Error : TON_TIME;
      lfb_TON_State : TON_TIME;
      lfb_F_Trig_ConveyerBelt : F_TRIG;
   END_VAR
BEGIN
   IF #lx_Init THEN

       // wait time state
       #lfb_TON_State(IN := NOT #lx_Start_TON_State,
                      PT := T#2s);

       // runtime monitoring error
       #lfb_TON_Error(IN := #lx_Time_Error,
                      PT := T#30s);

       // state of the MPO cyclically transmitted to the cloud
       IF (#lfb_TON_State.Q OR (#li_Lights <> #li_Lights_old)) AND NOT #lx_Start_TON_State THEN
           #li_Lights_old := #li_Lights;
           #lx_Start_TON_State := TRUE;
           #li_Return_LDT := RD_SYS_T(#ldt_MQTT);
           "gtyp_Interface_Dashboard".Subscribe.State_MPO.ldt_ts := DT_TO_LDT(#ldt_MQTT);
           "gtyp_Interface_Dashboard".Subscribe.State_MPO.i_code := #li_Lights;
           "gtyp_Interface_Dashboard".Subscribe.State_MPO.s_description := '';
           "gtyp_Interface_Dashboard".Subscribe.State_MPO.s_station := 'mpo';
           "gtyp_Interface_Dashboard".Subscribe.State_MPO.s_target := '';
       END_IF;

       // restart wait time state
       IF NOT #lfb_TON_State.Q AND #lx_Start_TON_State THEN
           #lx_Start_TON_State := FALSE;
       END_IF;

       // FB TON Wait
       #lfb_TON_Wait(IN := #lx_Start_TON_Wait,
                     PT := #lt_TON_Wait);

       // falling edge light barrier end of Conveyor Belt
       #lfb_F_Trig_ConveyerBelt(CLK := NOT "IX_MPO_LightBarrierEndOfConBelt_I3");

       //Run-on time Conveyer Belt
       #lfb_TOF_ConveyerBelt_Out(IN := #lfb_F_Trig_ConveyerBelt.Q,
                                 PT := T#5000ms);

       // FB blinker intervall 1s
       #lfb_blinker(int_periodendauer := T#1000ms);

       // step chain HBW
       CASE #li_StepCase OF

           0:  // init
               #lx_Start_TON_Wait := FALSE;
               #lx_Time_Error := FALSE;

               IF NOT "gtyp_MPO".x_Error AND NOT "gtyp_MPO".x_Start_Park_Position THEN
                   #li_StepCase := 10;
               END_IF;

           10: // turn-on Compressor and turn off oven light 
               #li_Lights := 2;
               "QX_MPO_LightOven_Q9" := FALSE;
               "QX_MPO_Compressor_Q10" := TRUE;

               #lx_Start_TON_Wait := TRUE;
               #lt_TON_Wait := T#500ms;

               IF #lfb_TON_Wait.Q THEN
                   #lx_Start_TON_Wait := FALSE;
                   #li_StepCase := 20;
               END_IF;

           20:  // Open oven door 
               "QX_MPO_ValveOvenDoor_Q13" := TRUE;
               "QX_MPO_ValveLowering_Q12" := FALSE;

               #lx_Start_TON_Wait := TRUE;
               #lt_TON_Wait := T#2000ms;

               IF #lfb_TON_Wait.Q THEN
                   #lx_Start_TON_Wait := FALSE;
                   #li_StepCase := 30;
               END_IF;

           30: // Position oven feeder retract
               IF "IX_MPO_RefSwitchOvenFeederOutside_I7" OR NOT "IX_MPO_RefSwitchOvenFeederInside_I6" THEN
                   "QX_MPO_M4_OvenFeederRetract_Q5" := TRUE;
                   "QX_MPO_M4_OvenFeederExtend_Q6" := FALSE;
               ELSIF NOT "IX_MPO_RefSwitchOvenFeederOutside_I7" AND "IX_MPO_RefSwitchOvenFeederInside_I6" THEN
                   "QX_MPO_M4_OvenFeederRetract_Q5" := FALSE;
                   "QX_MPO_M4_OvenFeederExtend_Q6" := FALSE;
                   #li_StepCase := 40;
               END_IF;

           40:  // Close door, Position Vacuum Towards Turn Table and vacuum off

               "QX_MPO_ValveOvenDoor_Q13" := FALSE;

               "QX_MPO_M5_VacuumTowardsTurnTable_Q8" := TRUE;
               "QX_MPO_M5_VacuumTowardsOven_Q7" := FALSE;
               "QX_MPO_ValveVacuum_Q11" := FALSE;

               IF "IX_MPO_RefSwitchVac_PosOven_I8" OR NOT "IX_MPO_RefSwitchVac_PosTurnTable_I5" THEN
                   "QX_MPO_M5_VacuumTowardsTurnTable_Q8" := TRUE;
                   "QX_MPO_M5_VacuumTowardsOven_Q7" := FALSE;
               ELSIF NOT "IX_MPO_RefSwitchVac_PosOven_I8" AND "IX_MPO_RefSwitchVac_PosTurnTable_I5" THEN
                   "QX_MPO_M5_VacuumTowardsTurnTable_Q8" := FALSE;
                   "QX_MPO_M5_VacuumTowardsOven_Q7" := FALSE;
                   #li_StepCase := 50;
               END_IF
               ;

           50: // saw, valve feeder conveyor belt off
               "QX_MPO_M3_Saw_Q4" := FALSE;
               "QX_MPO_ValveFeeder_Q14" := FALSE;
               "QX_MPO_M2_ConveyorBeltForward_Q3" := FALSE;

               IF "IX_MPO_RefSwitchTurnTable_PosSaw_I4" OR "IX_MPO_RefSwitchTurnTable_PosBelt_I2" OR NOT "IX_MPO_RefSwitchTurnTable_PosVac_I1" THEN
                   "QX_MPO_M1_TurnTableClockwise_Q1" := FALSE;
                   "QX_MPO_M1_TurnTableCounterclockwise_Q2" := TRUE;
               ELSIF NOT "IX_MPO_RefSwitchTurnTable_PosSaw_I4" AND NOT "IX_MPO_RefSwitchTurnTable_PosBelt_I2" AND "IX_MPO_RefSwitchTurnTable_PosVac_I1" THEN
                   "QX_MPO_M1_TurnTableClockwise_Q1" := FALSE;
                   "QX_MPO_M1_TurnTableCounterclockwise_Q2" := FALSE;
                   "QX_MPO_Compressor_Q10" := FALSE;
                   #li_StepCase := 60;
               END_IF;

           60: // wait for request discard form VGR
               #li_Lights := 1;
               IF "gtyp_VGR".x_MPO_Req_Discard THEN
                   #li_Lights := 2;
                   "QX_MPO_Compressor_Q10" := TRUE;
                   #li_StepCase := 70;
               END_IF;

           70: // wait sequence
               #lx_Start_TON_Wait := TRUE;
               #lt_TON_Wait := T#500ms;

               IF #lfb_TON_Wait.Q THEN
                   #lx_Start_TON_Wait := FALSE;
                   #li_StepCase := 80;
               END_IF;

           80: // open oven door
               "QX_MPO_ValveOvenDoor_Q13" := TRUE;

               #lx_Start_TON_Wait := TRUE;
               #lt_TON_Wait := T#2000ms;

               IF #lfb_TON_Wait.Q THEN
                   #lx_Start_TON_Wait := FALSE;
                   #li_StepCase := 90;
               END_IF;

           90: // oven feeder extend
               "QX_MPO_M4_OvenFeederRetract_Q5" := FALSE;
               "QX_MPO_M4_OvenFeederExtend_Q6" := TRUE;

               IF "IX_MPO_RefSwitchOvenFeederOutside_I7" AND NOT "IX_MPO_RefSwitchOvenFeederInside_I6" THEN
                   "QX_MPO_M4_OvenFeederRetract_Q5" := FALSE;
                   "QX_MPO_M4_OvenFeederExtend_Q6" := FALSE;
                   "gtyp_MPO".x_MPO_Discards_Accepted := FALSE;
                   "gtyp_MPO".x_Discard_Ready := TRUE;
                   #li_StepCase := 100;
               END_IF;

           100: // wait for VGR discard workpiece

               #lx_Time_Error := TRUE;

               IF "gtyp_VGR".x_MPO_Discards AND NOT "IX_MPO_LightBarrierOven_I9" THEN
                   "gtyp_Interface_Dashboard".Subscribe.State_MPO.x_active := TRUE;
                   "gtyp_MPO".History := "gtyp_VGR".History;
                   "gtyp_MPO".Workpiece := "gtyp_VGR".Workpiece;
                   "gtyp_MPO".x_Discard_Ready := FALSE;
                   "gtyp_MPO".x_MPO_Discards_Accepted := TRUE;
                   #lx_Time_Error := FALSE;
                   #li_StepCase := 105;
               END_IF;

               // runtime error
               IF #lfb_TON_Error.Q THEN
                   #li_Lights := 4;
                   #lx_Time_Error := FALSE;
                   "gtyp_Interface_Dashboard".Subscribe.State_Order.ldt_ts := DT_TO_LDT(#ldt_MQTT);
                   "gtyp_Interface_Dashboard".Subscribe.State_Order.s_state := 'WAITING_FOR_ORDER';
                   "gtyp_Interface_Dashboard".Subscribe.State_Order.s_type := '';
                   "gtyp_Interface_Dashboard".Subscribe.State_MPO.x_active := FALSE;
                   "gtyp_MPO".x_Discard_Ready := FALSE;
                   "gtyp_MPO".x_MPO_Discards_Accepted := FALSE;
                   "gtyp_MPO".x_Error := TRUE;
                   #li_StepCase := 0;
               END_IF;

           105: // VGR outside oven feeder - oven feeder retract
               IF NOT "gtyp_VGR".x_MPO_Discards AND "IX_MPO_RefSwitchOvenFeederOutside_I7" AND NOT "IX_MPO_RefSwitchOvenFeederInside_I6" THEN
                   "gtyp_MPO".x_MPO_Discards_Accepted := FALSE;
                   "QX_MPO_M4_OvenFeederRetract_Q5" := TRUE;
                   "QX_MPO_M4_OvenFeederExtend_Q6" := FALSE;
                   #li_StepCase := 110;
               END_IF;

           110: // sensor oven feeder inside reached
               IF NOT "IX_MPO_RefSwitchOvenFeederOutside_I7" AND "IX_MPO_RefSwitchOvenFeederInside_I6" THEN
                   "QX_MPO_M4_OvenFeederRetract_Q5" := FALSE;
                   "QX_MPO_M4_OvenFeederExtend_Q6" := FALSE;
                   #li_StepCase := 120;
               END_IF;

           120: // close oven door
               "QX_MPO_ValveOvenDoor_Q13" := FALSE;

               #lx_Start_TON_Wait := TRUE;
               #lt_TON_Wait := T#2000ms;

               IF #lfb_TON_Wait.Q THEN
                   #lx_Start_TON_Wait := FALSE;
                   #li_StepCase := 130;
               END_IF;

           130: // processing time flashing interval
               "QX_MPO_LightOven_Q9" := #lfb_blinker.outx_blinker;

               IF NOT "gtyp_VGR".x_MPO_Discards THEN
                   #li_Return_LDT := RD_SYS_T(#ldt_MQTT);
                   "gtyp_MPO".History[5].i_code := 500;
                   "gtyp_MPO".History[5].ldt_ts := DT_TO_LDT(#ldt_MQTT);

                   "QX_MPO_M5_VacuumTowardsOven_Q7" := TRUE;
                   "QX_MPO_M5_VacuumTowardsTurnTable_Q8" := FALSE;

                   IF NOT "IX_MPO_RefSwitchVac_PosTurnTable_I5" AND "IX_MPO_RefSwitchVac_PosOven_I8" THEN
                       "QX_MPO_M5_VacuumTowardsOven_Q7" := FALSE;
                       "QX_MPO_M5_VacuumTowardsTurnTable_Q8" := FALSE;
                   END_IF;
               END_IF;

               #lx_Start_TON_Wait := TRUE;
               #lt_TON_Wait := T#4000ms;

               IF #lfb_TON_Wait.Q THEN
                   #lx_Start_TON_Wait := FALSE;
                   #li_StepCase := 140;
               END_IF;

           140: // open oven door
               "QX_MPO_LightOven_Q9" := FALSE;
               "QX_MPO_ValveOvenDoor_Q13" := TRUE;

               IF NOT "gtyp_VGR".x_MPO_Discards THEN
                   "QX_MPO_M5_VacuumTowardsOven_Q7" := TRUE;
                   "QX_MPO_M5_VacuumTowardsTurnTable_Q8" := FALSE;

                   IF NOT "IX_MPO_RefSwitchVac_PosTurnTable_I5" AND "IX_MPO_RefSwitchVac_PosOven_I8" THEN
                       "QX_MPO_M5_VacuumTowardsOven_Q7" := FALSE;
                       "QX_MPO_M5_VacuumTowardsTurnTable_Q8" := FALSE;
                   END_IF;
               END_IF;

               #lx_Start_TON_Wait := TRUE;
               #lt_TON_Wait := T#2000ms;

               IF #lfb_TON_Wait.Q THEN
                   #lx_Start_TON_Wait := FALSE;
                   #li_StepCase := 150;
               END_IF;

           150: // oven feeder extend

               "QX_MPO_M4_OvenFeederRetract_Q5" := FALSE;
               "QX_MPO_M4_OvenFeederExtend_Q6" := TRUE;

               IF NOT "gtyp_VGR".x_MPO_Discards THEN
                   "QX_MPO_M5_VacuumTowardsOven_Q7" := TRUE;
                   "QX_MPO_M5_VacuumTowardsTurnTable_Q8" := FALSE;

                   IF NOT "IX_MPO_RefSwitchVac_PosTurnTable_I5" AND "IX_MPO_RefSwitchVac_PosOven_I8" THEN
                       "QX_MPO_M5_VacuumTowardsOven_Q7" := FALSE;
                       "QX_MPO_M5_VacuumTowardsTurnTable_Q8" := FALSE;
                   END_IF;
               END_IF;

               IF "IX_MPO_RefSwitchOvenFeederOutside_I7" AND NOT "IX_MPO_RefSwitchOvenFeederInside_I6" THEN
                   "QX_MPO_M4_OvenFeederRetract_Q5" := FALSE;
                   "QX_MPO_M4_OvenFeederExtend_Q6" := FALSE;
               END_IF;

               IF "IX_MPO_RefSwitchOvenFeederOutside_I7" AND NOT "IX_MPO_RefSwitchOvenFeederInside_I6"
                   AND NOT "IX_MPO_RefSwitchVac_PosTurnTable_I5" AND "IX_MPO_RefSwitchVac_PosOven_I8" THEN
                   "QX_MPO_M5_VacuumTowardsOven_Q7" := FALSE;
                   "QX_MPO_M5_VacuumTowardsTurnTable_Q8" := FALSE;
                   "QX_MPO_M4_OvenFeederRetract_Q5" := FALSE;
                   "QX_MPO_M4_OvenFeederExtend_Q6" := FALSE;
                   #li_StepCase := 160;
               END_IF;

           160: // vacuum suction device down
               "QX_MPO_ValveLowering_Q12" := TRUE;

               #lx_Start_TON_Wait := TRUE;
               #lt_TON_Wait := T#1000ms;

               IF #lfb_TON_Wait.Q THEN
                   #lx_Start_TON_Wait := FALSE;
                   #li_StepCase := 170;
               END_IF;

           170: // vacuum suction device picks up the workpiece
               "QX_MPO_ValveVacuum_Q11" := TRUE;

               #lx_Start_TON_Wait := TRUE;
               #lt_TON_Wait := T#1000ms;

               IF #lfb_TON_Wait.Q THEN
                   #lx_Start_TON_Wait := FALSE;
                   #li_StepCase := 180;
               END_IF;

           180: // vacuum suction device up
               "QX_MPO_ValveLowering_Q12" := FALSE;

               #lx_Start_TON_Wait := TRUE;
               #lt_TON_Wait := T#1000ms;

               IF #lfb_TON_Wait.Q THEN
                   #lx_Start_TON_Wait := FALSE;
                   #li_StepCase := 190;
               END_IF;

           190: // oven feeder retract and vacuum towards turn table
               "QX_MPO_M4_OvenFeederRetract_Q5" := TRUE;
               "QX_MPO_M4_OvenFeederExtend_Q6" := FALSE;
               "QX_MPO_M5_VacuumTowardsOven_Q7" := FALSE;
               "QX_MPO_M5_VacuumTowardsTurnTable_Q8" := TRUE;

               IF "IX_MPO_RefSwitchVac_PosTurnTable_I5" AND NOT "IX_MPO_RefSwitchVac_PosOven_I8" THEN
                   "QX_MPO_M5_VacuumTowardsOven_Q7" := FALSE;
                   "QX_MPO_M5_VacuumTowardsTurnTable_Q8" := FALSE;
               END_IF;

               IF NOT "IX_MPO_RefSwitchOvenFeederOutside_I7" AND "IX_MPO_RefSwitchOvenFeederInside_I6" THEN
                   "QX_MPO_M4_OvenFeederRetract_Q5" := FALSE;
                   "QX_MPO_M4_OvenFeederExtend_Q6" := FALSE;
               END_IF;

               IF NOT "IX_MPO_RefSwitchOvenFeederOutside_I7" AND "IX_MPO_RefSwitchOvenFeederInside_I6"
                   AND "IX_MPO_RefSwitchVac_PosTurnTable_I5" AND NOT "IX_MPO_RefSwitchVac_PosOven_I8" THEN
                   "QX_MPO_M5_VacuumTowardsOven_Q7" := FALSE;
                   "QX_MPO_M5_VacuumTowardsTurnTable_Q8" := FALSE;
                   "QX_MPO_M4_OvenFeederRetract_Q5" := FALSE;
                   "QX_MPO_M4_OvenFeederExtend_Q6" := FALSE;
                   "QX_MPO_ValveOvenDoor_Q13" := FALSE;
                   #li_StepCase := 200;
               END_IF;

           200: // vacuum suction device down at turn table
               IF "IX_MPO_RefSwitchTurnTable_PosVac_I1" THEN
                   "QX_MPO_ValveLowering_Q12" := TRUE;

                   #lx_Start_TON_Wait := TRUE;
                   #lt_TON_Wait := T#2000ms;

                   IF #lfb_TON_Wait.Q THEN
                       #lx_Start_TON_Wait := FALSE;
                       #li_StepCase := 210;
                   END_IF;
               END_IF;

           210: // vacuum off
               "QX_MPO_ValveVacuum_Q11" := FALSE;

               #lx_Start_TON_Wait := TRUE;
               #lt_TON_Wait := T#2000ms;

               IF #lfb_TON_Wait.Q THEN
                   #lx_Start_TON_Wait := FALSE;
                   #li_StepCase := 220;
               END_IF;

           220: // vacuum suction device up
               "QX_MPO_ValveLowering_Q12" := FALSE;

               #lx_Start_TON_Wait := TRUE;
               #lt_TON_Wait := T#2000ms;

               IF #lfb_TON_Wait.Q THEN
                   #lx_Start_TON_Wait := FALSE;
                   #li_StepCase := 230;
               END_IF;

           230: // Position turn table saw
               IF NOT "IX_MPO_RefSwitchTurnTable_PosSaw_I4" AND NOT "IX_MPO_RefSwitchTurnTable_PosBelt_I2" AND "IX_MPO_RefSwitchTurnTable_PosVac_I1" THEN
                   "QX_MPO_M1_TurnTableClockwise_Q1" := TRUE;
                   "QX_MPO_M1_TurnTableCounterclockwise_Q2" := FALSE;
               ELSIF "IX_MPO_RefSwitchTurnTable_PosSaw_I4" OR "IX_MPO_RefSwitchTurnTable_PosBelt_I2" AND NOT "IX_MPO_RefSwitchTurnTable_PosVac_I1" THEN
                   "QX_MPO_M1_TurnTableClockwise_Q1" := FALSE;
                   "QX_MPO_M1_TurnTableCounterclockwise_Q2" := FALSE;
                   #li_StepCase := 240;
               END_IF;

           240: // Start sawing
               "QX_MPO_M3_Saw_Q4" := TRUE;

               #lx_Start_TON_Wait := TRUE;
               #lt_TON_Wait := T#4000ms;

               IF #lfb_TON_Wait.Q THEN
                   #li_Return_LDT := RD_SYS_T(#ldt_MQTT);
                   "gtyp_MPO".History[6].i_code := 600;
                   "gtyp_MPO".History[6].ldt_ts := DT_TO_LDT(#ldt_MQTT);

                   #lx_Start_TON_Wait := FALSE;
                   "QX_MPO_M3_Saw_Q4" := FALSE;
                   #li_StepCase := 250;
               END_IF;

           250: // Position turn table Pos Belt
               IF "IX_MPO_RefSwitchTurnTable_PosSaw_I4" AND NOT "IX_MPO_RefSwitchTurnTable_PosBelt_I2" AND NOT "IX_MPO_RefSwitchTurnTable_PosVac_I1" THEN
                   "QX_MPO_M1_TurnTableClockwise_Q1" := TRUE;
                   "QX_MPO_M1_TurnTableCounterclockwise_Q2" := FALSE;
               ELSIF NOT "IX_MPO_RefSwitchTurnTable_PosSaw_I4" AND "IX_MPO_RefSwitchTurnTable_PosBelt_I2" AND NOT "IX_MPO_RefSwitchTurnTable_PosVac_I1" THEN
                   "QX_MPO_M1_TurnTableClockwise_Q1" := FALSE;
                   "QX_MPO_M1_TurnTableCounterclockwise_Q2" := FALSE;
                   #li_StepCase := 260;
               END_IF;

           260: // put workpiece to belt
               "QX_MPO_ValveFeeder_Q14" := TRUE;

               #lx_Start_TON_Wait := TRUE;
               #lt_TON_Wait := T#1000ms;

               IF #lfb_TON_Wait.Q THEN
                   #lx_Start_TON_Wait := FALSE;
                   "QX_MPO_ValveFeeder_Q14" := FALSE;
                   "QX_MPO_Compressor_Q10" := FALSE;
                   #li_StepCase := 270;
               END_IF;

           270: // Position turn table Pos Vacuum
               IF "IX_MPO_RefSwitchTurnTable_PosSaw_I4" OR "IX_MPO_RefSwitchTurnTable_PosBelt_I2" OR NOT "IX_MPO_RefSwitchTurnTable_PosVac_I1" THEN
                   "QX_MPO_M1_TurnTableClockwise_Q1" := FALSE;
                   "QX_MPO_M1_TurnTableCounterclockwise_Q2" := TRUE;
               ELSIF NOT "IX_MPO_RefSwitchTurnTable_PosSaw_I4" AND NOT "IX_MPO_RefSwitchTurnTable_PosBelt_I2" AND "IX_MPO_RefSwitchTurnTable_PosVac_I1" THEN
                   "QX_MPO_M1_TurnTableClockwise_Q1" := FALSE;
                   "QX_MPO_M1_TurnTableCounterclockwise_Q2" := FALSE;
                   "QX_MPO_Compressor_Q10" := FALSE;
                   #li_StepCase := 280;
               END_IF;

           280: // Start conveyor belt
               "QX_MPO_M2_ConveyorBeltForward_Q3" := TRUE;

               #lx_Time_Error := TRUE;

               IF #lfb_TOF_ConveyerBelt_Out.Q THEN
                   "gtyp_SLD".History := "gtyp_MPO".History;
                   "gtyp_SLD".Workpiece := "gtyp_MPO".Workpiece;
                   "gtyp_MPO".Workpiece.s_id := '0';
                   "gtyp_MPO".Workpiece.s_state := '';
                   "gtyp_MPO".Workpiece.s_type := '';
                   FOR #li_Counter := 1 TO 8 DO
                       "gtyp_MPO".History[#li_Counter].i_code := 0;
                       "gtyp_MPO".History[#li_Counter].ldt_ts := DT#1990-01-01-00:00:00;
                   END_FOR;

                   "gtyp_Interface_Dashboard".Subscribe.State_MPO.x_active := FALSE;

                   #lx_Time_Error := FALSE;
                   #li_StepCase := 290;
               END_IF;

               // runtime error
               IF #lfb_TON_Error.Q THEN
                   #li_Lights := 4;
                   #lx_Time_Error := FALSE;
                   "QX_MPO_M2_ConveyorBeltForward_Q3" := FALSE;
                   "gtyp_Interface_Dashboard".Subscribe.State_MPO.x_active := FALSE;
                   "gtyp_MPO".x_Error := TRUE;
                   #li_StepCase := 0;
               END_IF;

           290: // wait for runtime on conveyor belt

               IF NOT #lfb_TOF_ConveyerBelt_Out.Q THEN
                   #lx_Start_TON_Wait := FALSE;
                   "QX_MPO_M2_ConveyorBeltForward_Q3" := FALSE;
                   #li_StepCase := 60;
               END_IF;
               // Statement section ELSE
           ELSE
               ;
       END_CASE;

       "QW_MPO_PWM_TurnTable_M1" := "gtyp_MPO"."i_PWM_TurnTable";
       "QW_MPO_PWM_Vacuum_M5" := "gtyp_MPO"."i_PWM_Vacuum";

   ELSE
       #li_Lights := 1;
       #lx_Init := TRUE;
       "gtyp_MPO".x_Start_Park_Position := FALSE;
       "gtyp_MPO".x_Park_Position_Reached := FALSE;
   END_IF;
END_FUNCTION_BLOCK

FUNCTION_BLOCK "PRG_MPO_Set_Park_Position"   // FB39, SCL
TITLE = Program Set Positioning HBW
{ S7_Optimized_Access := 'TRUE' }
AUTHOR : A.Schaefer
VERSION : 0.0
   VAR
      lx_Init : Bool;
      lx_Start_TON_Wait : Bool;
      lt_TON_Wait : Time;
      li_StepCase : Int;
      lfb_TON_Wait : TON_TIME;
      lfb_R_Trig_Start_Park_Pos : R_TRIG;
   END_VAR
BEGIN
   IF #lx_Init THEN

       // FB TON Wait
       #lfb_TON_Wait(IN := #lx_Start_TON_Wait,
                     PT := #lt_TON_Wait);

       #lfb_R_Trig_Start_Park_Pos(CLK := "gtyp_Setup".x_Park_Position
                                  OR "IX_Set_Park_Position");

       // Set Start Park Position   
       IF #lfb_R_Trig_Start_Park_Pos.Q THEN
           "gtyp_MPO".x_Start_Park_Position := TRUE;
           #li_StepCase := 0;
       END_IF;

       // not Start Park Pos Step 0
       IF NOT "gtyp_MPO".x_Start_Park_Position THEN
           #li_StepCase := 0;
       END_IF;

       // step chain HBW
       CASE #li_StepCase OF

           0:  // init
               #lx_Start_TON_Wait := FALSE;
               #li_StepCase := 10;

           10:  // Set Positioning activ?
               IF "gtyp_MPO".x_Start_Park_Position AND NOT "gtyp_MPO".x_Park_Position_Reached THEN
                   #li_StepCase := 20;
               END_IF;

           20: // Towards
               "QX_MPO_M5_VacuumTowardsTurnTable_Q8" := FALSE;
               "QX_MPO_M5_VacuumTowardsOven_Q7" := TRUE;
               #lx_Start_TON_Wait := TRUE;
               #lt_TON_Wait := T#4000ms;

               IF #lfb_TON_Wait.Q THEN
                   "QX_MPO_M5_VacuumTowardsTurnTable_Q8" := FALSE;
                   "QX_MPO_M5_VacuumTowardsOven_Q7" := FALSE;
                   #lx_Start_TON_Wait := FALSE;
                   #li_StepCase := 30;
               END_IF;

           30: // homing vertical axis
               "QX_MPO_M1_TurnTableClockwise_Q1" := TRUE;
               "QX_MPO_M1_TurnTableCounterclockwise_Q2" := FALSE;
               #lx_Start_TON_Wait := TRUE;
               #lt_TON_Wait := T#1000ms;

               IF #lfb_TON_Wait.Q THEN
                   "QX_MPO_M1_TurnTableClockwise_Q1" := FALSE;
                   "QX_MPO_M1_TurnTableCounterclockwise_Q2" := FALSE;
                   #lx_Start_TON_Wait := FALSE;
                   #li_StepCase := 40;
               END_IF;

           40: // Deciding which doing
               "gtyp_MPO".x_Park_Position_Reached := TRUE;


               // Statement section ELSE    
           ELSE
               ;
       END_CASE;

   ELSE
       #lx_Init := TRUE;
   END_IF;
END_FUNCTION_BLOCK

// folder: 3.4. SLD

FUNCTION_BLOCK "PRG_SLD_Ablauf"   // FB19, SCL
TITLE = Program Ablauf SLD
{ S7_Optimized_Access := 'TRUE' }
AUTHOR : A.Schaefer
VERSION : 0.0
   VAR
      lx_Init : Bool;
      lx_Start_TON_Wait : Bool;
      lx_Time_Error : Bool;
      lt_TON_Wait : Time;
      lx_Start_TON_State : Bool;
      ldt_MQTT : Date_And_Time;
      li_Return_LDT : Int;
      li_Lights : Int;
      li_Lights_old : Int;
      lw_ColorValueMin : Word;
      li_CounterActual : Int;
      lx_White : Bool;
      lx_Blue : Bool;
      lx_Red : Bool;
      li_StepCase : Int;
      ls_Color : String;
      lfb_TOF_ConveyerBelt_Out : TOF_TIME;
      lfb_TON_Wait : TON_TIME;
      lfb_TON_Error : TON_TIME;
      lfb_TON_State : TON_TIME;
      lfb_F_Trig_Counter : F_TRIG;
      lfb_R_Trig_Counter : R_TRIG;
   END_VAR
BEGIN
   IF #lx_Init THEN

       // Restart after set Positioning
       IF "gtyp_Setup".x_Color_Sensor_Calibration THEN
           #li_StepCase := 0;
       END_IF;

       // wait time state
       #lfb_TON_State(IN := NOT #lx_Start_TON_State,
                      PT := T#2s);

       // state of the SLD cyclically transmitted to the cloud
       IF (#lfb_TON_State.Q OR (#li_Lights <> #li_Lights_old)) AND NOT #lx_Start_TON_State THEN
           #li_Lights_old := #li_Lights;
           #lx_Start_TON_State := TRUE;
           #li_Return_LDT := RD_SYS_T(#ldt_MQTT);
           "gtyp_Interface_Dashboard".Subscribe.State_SLD.ldt_ts := DT_TO_LDT(#ldt_MQTT);
           "gtyp_Interface_Dashboard".Subscribe.State_SLD.i_code := #li_Lights;
           "gtyp_Interface_Dashboard".Subscribe.State_SLD.s_description := '';
           "gtyp_Interface_Dashboard".Subscribe.State_SLD.s_station := 'sld';
           "gtyp_Interface_Dashboard".Subscribe.State_SLD.s_target := '';
       END_IF;

       // restart wait time state
       IF NOT #lfb_TON_State.Q AND #lx_Start_TON_State THEN
           #lx_Start_TON_State := FALSE;
       END_IF;

       // FB TON Wait
       #lfb_TON_Wait(IN := #lx_Start_TON_Wait,
                     PT := #lt_TON_Wait);

       // runtime monitoring error
       #lfb_TON_Error(IN := #lx_Time_Error,
                      PT := T#30s);

       // rising edge pulse counter
       #lfb_R_Trig_Counter(CLK := "IX_SLD_PulseCounter_I1");

       // falling edge pulse counter
       #lfb_F_Trig_Counter(CLK := "IX_SLD_PulseCounter_I1");

       // step chain SLD
       CASE #li_StepCase OF

           0:  // Init
               #lx_Start_TON_Wait := FALSE;
               #lx_Time_Error := FALSE;
               #li_Lights := 1;

               IF NOT "gtyp_SLD".x_Error AND NOT "gtyp_Setup".x_Color_Sensor_Calibration THEN
                   #li_StepCase := 10;
               END_IF;

           10: // turn-on Compressor and wait sequence 
               #li_Lights := 2;
               "QX_SLD_Compressor_Q2" := TRUE;

               #lx_Start_TON_Wait := TRUE;
               #lt_TON_Wait := T#1000ms;

               IF #lfb_TON_Wait.Q THEN
                   #lx_Start_TON_Wait := FALSE;
                   #li_StepCase := 20;
               END_IF;

           20:  // reset Ejectors
               "QX_SLD_ValveFirstEjectorWhite_Q3" := FALSE;
               "QX_SLD_ValveSecondEjectorRed_Q4" := FALSE;
               "QX_SLD_ValveThirdEjectorBlue_Q5" := FALSE;
               "QX_SLD_M1_ConveyorBelt_Q1" := FALSE;

               #lx_Start_TON_Wait := TRUE;
               #lt_TON_Wait := T#2000ms;

               IF #lfb_TON_Wait.Q THEN
                   #lx_Start_TON_Wait := FALSE;
                   #li_StepCase := 30;
               END_IF;

           30: // turn-off Compressor 

               "QX_SLD_Compressor_Q2" := FALSE;

               #li_StepCase := 40;

           40: // start belt if Light barrier I2 active

               #li_Lights := 1;
               IF NOT "IX_SLD_LightBarrierInlet_I2" THEN
                   "gtyp_Interface_Dashboard".Subscribe.State_SLD.x_active := TRUE;
                   #li_Lights := 2;
                   "QX_SLD_Compressor_Q2" := TRUE;
                   "QX_SLD_M1_ConveyorBelt_Q1" := TRUE;
                   #lw_ColorValueMin := 40000;
                   #li_CounterActual := 0;
                   #lx_Blue := FALSE;
                   #lx_Red := FALSE;
                   #lx_White := FALSE;
                   #li_StepCase := 50;
               END_IF;

           50: // take the min Value of the Color sensor
               IF #lw_ColorValueMin > "IW_SLD_ColorSensor_A4" THEN
                   #lw_ColorValueMin := "IW_SLD_ColorSensor_A4";
               END_IF;

               #lx_Time_Error := TRUE;

               // Stop when light barrier I3 on 
               IF NOT "IX_SLD_LightBarrierBehindColorSensor_I3" THEN
                   #lx_Time_Error := FALSE;
                   #li_StepCase := 60;
               END_IF;

               // runtime error
               IF #lfb_TON_Error.Q THEN
                   #li_Lights := 4;
                   #lx_Time_Error := FALSE;
                   "QX_SLD_Compressor_Q2" := FALSE;
                   "QX_SLD_M1_ConveyorBelt_Q1" := FALSE;
                   "gtyp_Interface_Dashboard".Subscribe.State_SLD.x_active := FALSE;
                   "gtyp_SLD".x_Error := TRUE;
                   #li_StepCase := 0;
               END_IF;

           60: // analyze color

               IF #lw_ColorValueMin >= "gtyp_SLD".w_Threshold_Red_Blue THEN
                   #lx_Blue := TRUE;
               ELSIF #lw_ColorValueMin <= "gtyp_SLD".w_Threshold_White_Red THEN
                   #lx_White := TRUE;
               ELSIF #lw_ColorValueMin > "gtyp_SLD".w_Threshold_White_Red AND #lw_ColorValueMin < "gtyp_SLD".w_Threshold_Red_Blue THEN
                   #lx_Red := TRUE;
               END_IF;

               // actual counter
               IF #lfb_R_Trig_Counter.Q OR #lfb_F_Trig_Counter.Q THEN
                   #li_CounterActual := #li_CounterActual + 1;
               END_IF;

               // Reached counter value and color set Ejector
               IF (#li_CounterActual = "gtyp_SLD".i_CounterValue_Blue) AND #lx_Blue THEN
                   "QX_SLD_ValveThirdEjectorBlue_Q5" := TRUE;
                   #li_Return_LDT := RD_SYS_T(#ldt_MQTT);
                   "gtyp_SLD".Workpiece.s_state := 'PROCESSED';
                   "gtyp_SLD".History[7].i_code := 700;
                   "gtyp_SLD".History[7].ldt_ts := DT_TO_LDT(#ldt_MQTT);
                   #li_StepCase := 70;
               ELSIF (#li_CounterActual = "gtyp_SLD".i_CounterValue_White) AND #lx_White THEN
                   "QX_SLD_ValveFirstEjectorWhite_Q3" := TRUE;
                   #li_Return_LDT := RD_SYS_T(#ldt_MQTT);
                   "gtyp_SLD".Workpiece.s_state := 'PROCESSED';
                   "gtyp_SLD".History[7].i_code := 700;
                   "gtyp_SLD".History[7].ldt_ts := DT_TO_LDT(#ldt_MQTT);
                   #li_StepCase := 70;
               ELSIF (#li_CounterActual = "gtyp_SLD".i_CounterValue_Red) AND #lx_Red THEN
                   "QX_SLD_ValveSecondEjectorRed_Q4" := TRUE;
                   #li_Return_LDT := RD_SYS_T(#ldt_MQTT);
                   "gtyp_SLD".Workpiece.s_state := 'PROCESSED';
                   "gtyp_SLD".History[7].i_code := 700;
                   "gtyp_SLD".History[7].ldt_ts := DT_TO_LDT(#ldt_MQTT);
                   #li_StepCase := 70;
               ELSIF (#li_CounterActual = 80) THEN
                   #li_Lights := 4;
                   "gtyp_SLD".x_Error := TRUE;
                   #li_StepCase := 70;
               END_IF;

           70: // wait sequence
               #lx_Start_TON_Wait := TRUE;
               #lt_TON_Wait := T#500ms;

               IF #lfb_TON_Wait.Q THEN
                   "QX_SLD_ValveThirdEjectorBlue_Q5" := FALSE;
                   "QX_SLD_ValveFirstEjectorWhite_Q3" := FALSE;
                   "QX_SLD_ValveSecondEjectorRed_Q4" := FALSE;
                   #lx_Start_TON_Wait := FALSE;
                   #li_StepCase := 80;
               END_IF;

           80: // wait sequence

               #lx_Start_TON_Wait := TRUE;
               #lt_TON_Wait := T#2000ms;

               IF #lfb_TON_Wait.Q THEN
                   "QX_SLD_Compressor_Q2" := FALSE;
                   #lx_Start_TON_Wait := FALSE;
                   #li_StepCase := 90;
               END_IF;

           90: // Stop belt
               "QX_SLD_M1_ConveyorBelt_Q1" := FALSE;
               #li_StepCase := 40;
               // Statement section ELSE
           ELSE
               ;
       END_CASE;

   ELSE
       "gtyp_SLD".x_Error := FALSE;
       #li_Lights := 1;
       #lx_Init := TRUE;
   END_IF;
END_FUNCTION_BLOCK

FUNCTION_BLOCK "PRG_SLD_Calibration_Color"   // FB33, SCL
TITLE = Program Calibration Color Sensor SLD
{ S7_Optimized_Access := 'TRUE' }
AUTHOR : A.Schaefer
VERSION : 0.0
   VAR
      lx_Init : Bool;
      lx_Start_TON_Wait : Bool;
      lx_Start_Positioning_m : Bool;
      lt_TON_Wait : Time;
      li_StepCase : Int;
      lw_ColorValueMin : Word;
      ldi_Pos_Horizontal : DInt;
      ldi_Pos_Vertical : DInt;
      lfb_R_Trig_Deaktivate : R_TRIG;
      lfb_TON_Wait : TON_TIME;
   END_VAR
BEGIN
   IF #lx_Init THEN

       // FB TON Wait
       #lfb_TON_Wait(IN := #lx_Start_TON_Wait,
                     PT := #lt_TON_Wait);

       #lfb_R_Trig_Deaktivate(CLK := NOT "gtyp_Setup".x_Color_Sensor_Calibration
                              OR NOT ("gtyp_Setup".i_Color_Sensor_Selection = 2));
       // Deaktivate step 0   
       IF #lfb_R_Trig_Deaktivate.Q THEN
           "gtyp_Setup".x_Calculate_Value_Color := FALSE;
           "gtyp_Setup".x_Set_Calib_Value_Color_Blue := FALSE;
           "gtyp_Setup".x_Set_Calib_Value_Color_Red := FALSE;
           "gtyp_Setup".x_Set_Calib_Value_Color_White := FALSE;
           "gtyp_Setup".w_Calib_ColorValue_Blue := 0;
           "gtyp_Setup".w_Calib_ColorValue_Red := 0;
           "gtyp_Setup".w_Calib_ColorValue_White := 0;
           "gtyp_Setup".w_Threshold_Red_Blue := 0;
           "gtyp_Setup".w_Threshold_White_Red := 0;
           "QX_SLD_M1_ConveyorBelt_Q1" := FALSE;
           #lw_ColorValueMin := 16#FF;
           #li_StepCase := 0;
       END_IF;

       // step chain HBW
       CASE #li_StepCase OF

           0:  // init
               #lx_Start_TON_Wait := FALSE;
               #li_StepCase := 10;

           10:  // Set Calibration activ?
               IF "gtyp_Setup".x_Color_Sensor_Calibration
                   AND ("gtyp_Setup".i_Color_Sensor_Selection = 2) THEN
                   "gtyp_Setup".x_Calculate_Value_Color := FALSE;
                   "gtyp_Setup".x_Set_Calib_Value_Color_Blue := FALSE;
                   "gtyp_Setup".x_Set_Calib_Value_Color_Red := FALSE;
                   "gtyp_Setup".x_Set_Calib_Value_Color_White := FALSE;
                   "gtyp_Setup".w_Calib_ColorValue_Blue := 0;
                   "gtyp_Setup".w_Calib_ColorValue_Red := 0;
                   "gtyp_Setup".w_Calib_ColorValue_White := 0;
                   "gtyp_Setup".w_Threshold_Red_Blue := 0;
                   "gtyp_Setup".w_Threshold_White_Red := 0;
                   "QX_SLD_M1_ConveyorBelt_Q1" := FALSE;
                   #lw_ColorValueMin := 16#FFFF;
                   #li_StepCase := 20;
               END_IF;

           20: // wait for set Values or Calculate

               IF NOT "IX_SLD_LightBarrierInlet_I2" THEN
                   "QX_SLD_M1_ConveyorBelt_Q1" := TRUE;
                   #lw_ColorValueMin := 16#FFFF;
               END_IF;

               IF #lw_ColorValueMin > "IW_SLD_ColorSensor_A4" THEN
                   #lw_ColorValueMin := "IW_SLD_ColorSensor_A4";
               END_IF;

               IF NOT "IX_SLD_LightBarrierBehindColorSensor_I3" THEN
                   "QX_SLD_M1_ConveyorBelt_Q1" := FALSE;
               END_IF;

               // Start new Positioning
               IF "gtyp_Setup".x_Set_Calib_Value_Color_Blue THEN
                   "gtyp_Setup".w_Calib_ColorValue_Blue := #lw_ColorValueMin;
                   "gtyp_Setup".x_Set_Calib_Value_Color_Blue := FALSE;
               ELSIF "gtyp_Setup".x_Set_Calib_Value_Color_Red THEN
                   "gtyp_Setup".w_Calib_ColorValue_Red := #lw_ColorValueMin;
                   "gtyp_Setup".x_Set_Calib_Value_Color_Red := FALSE;
               ELSIF "gtyp_Setup".x_Set_Calib_Value_Color_White THEN
                   "gtyp_Setup".w_Calib_ColorValue_White := #lw_ColorValueMin;
                   "gtyp_Setup".x_Set_Calib_Value_Color_White := FALSE;
               END_IF;

               "gtyp_Setup".w_Threshold_White_Red := "gtyp_Setup".w_Calib_ColorValue_White + (("gtyp_Setup".w_Calib_ColorValue_Red - "gtyp_Setup".w_Calib_ColorValue_White) / 2);
               "gtyp_Setup".w_Threshold_Red_Blue := "gtyp_Setup".w_Calib_ColorValue_Red + (("gtyp_Setup".w_Calib_ColorValue_Blue - "gtyp_Setup".w_Calib_ColorValue_Red) / 2);

               IF "gtyp_Setup".x_Calculate_Value_Color THEN
                   "gtyp_SLD".w_Threshold_White_Red := "gtyp_Setup".w_Threshold_White_Red;
                   "gtyp_SLD".w_Threshold_Red_Blue := "gtyp_Setup".w_Threshold_Red_Blue;
                   "gtyp_Setup".x_Calculate_Value_Color := FALSE;
               END_IF;

               // Statement section ELSE    
           ELSE
               ;
       END_CASE;

       IF ("gtyp_Setup".i_Color_Sensor_Selection = 2) THEN
           // Reload Pos Value
           "gtyp_Setup".w_Actual_ColorValue := "IW_SLD_ColorSensor_A4";
       END_IF;
   ELSE
       #lx_Init := TRUE;
   END_IF;
END_FUNCTION_BLOCK

FUNCTION_BLOCK "PRG_SLD_Set_Counter_Values"   // FB34, SCL
TITLE = Program Set counter Values SLD
{ S7_Optimized_Access := 'TRUE' }
AUTHOR : A.Schaefer
VERSION : 0.0
   VAR
      lx_Init : Bool;
      lfb_R_Trig_Calib_activ : R_TRIG;
   END_VAR
BEGIN
   IF #lx_Init THEN

       // Reload act. Counter Values
       IF NOT "gtyp_Setup".x_Counter_Value_Calibration THEN
           "gtyp_Setup".i_Calib_CounterValue_Blue := "gtyp_SLD".i_CounterValue_Blue;
           "gtyp_Setup".i_Calib_CounterValue_Red := "gtyp_SLD".i_CounterValue_Red;
           "gtyp_Setup".i_Calib_CounterValue_White := "gtyp_SLD".i_CounterValue_White;
       END_IF;

       // Set Counter Values   
       IF "gtyp_Setup".x_Set_CounterValues AND "gtyp_Setup".x_Counter_Value_Calibration THEN
           "gtyp_SLD".i_CounterValue_Blue := "gtyp_Setup".i_Calib_CounterValue_Blue;
           "gtyp_SLD".i_CounterValue_Red := "gtyp_Setup".i_Calib_CounterValue_Red;
           "gtyp_SLD".i_CounterValue_White := "gtyp_Setup".i_Calib_CounterValue_White;
           "gtyp_Setup".x_Set_CounterValues := FALSE;
       END_IF;

   ELSE
       #lx_Init := TRUE;
   END_IF;
END_FUNCTION_BLOCK

// folder: 3.5. SSC

FUNCTION_BLOCK "PRG_SSC_Axis_Vertical"   // FB11, SCL
TITLE = Program Axis vertical SSC
{ S7_Optimized_Access := 'TRUE' }
AUTHOR : A.Schaefer
VERSION : 0.0
   VAR
      lx_Init : Bool;
      lfb_Vertical_Axis : "FB_Axis";
   END_VAR
BEGIN
   IF #lx_Init THEN

       // FB Axis vertical
       #lfb_Vertical_Axis(ini_Axis := 5,
                          indi_Increment := "gtyp_SSC".Vertical_Axis.di_Increment,
                          inx_Ref_Switch := "IX_SSC_RefSwitchVerticalAxis_I1",
                          inx_Referencing := "gtyp_SSC".Vertical_Axis.x_Reference,
                          inx_Start_Positioning := "gtyp_SSC".Vertical_Axis.x_Start_Positioning,
                          indi_Target_Position := "gtyp_SSC".Vertical_Axis.di_Target_Position,
                          ini_PWM := "gtyp_SSC".Vertical_Axis.i_PWM,
                          inouttyp_Config := "gtyp_SSC".Vertical_Axis.Config,
                          inouttyp_Setup := "gtyp_SetupAxis");

       "QX_SSC_M1_VerticalAxisUp_Q1" := #lfb_Vertical_Axis.outx_Motor_Pos;
       "QX_SSC_M1_VerticalAxisDown_Q2" := #lfb_Vertical_Axis.outx_Motor_Neg;
       "QW_SSC_PWM_Vertical_M1" := #lfb_Vertical_Axis.outi_Motor_PWM;
       "gtyp_SSC".Vertical_Axis.di_Actual_Position := #lfb_Vertical_Axis.outdi_Actual_Position;
       "gtyp_SSC".Vertical_Axis.x_Referenced := #lfb_Vertical_Axis.outx_Referenced;
       "gtyp_SSC".Vertical_Axis.x_Position_Reached := #lfb_Vertical_Axis.outx_Position_Reached;
   ELSE
       #lx_Init := TRUE;
   END_IF;
END_FUNCTION_BLOCK

FUNCTION_BLOCK "PRG_SSC_Ablauf"   // FB12, SCL
TITLE = Program Ablauf SSC
{ S7_Optimized_Access := 'TRUE' }
AUTHOR : A.Schaefer
VERSION : 0.0
   VAR
      lx_Init : Bool;
      lx_FirstCentre : Bool;
      lx_Start : Bool;
      lx_Start_TON_State : Bool;
      lt_TON_Wait : Time;
      li_StepCase : Int;
      ldi_TargetPosition_Horizontal : DInt;
      ldi_TargetPosition_Vertical : DInt;
      lldt_ts_old : LDT;
      ldt_write : Date_And_Time;
      li_Return_write : Int;
      ldt_MQTT : Date_And_Time;
      li_Return_LDT : Int;
      lx_Start_TON_Wait : Bool;
      ldi_StepHorizontal : DInt;
      ldi_StepVertical : DInt;
      lfb_TON_Wait : TON_TIME;
      lfb_TON_State : TON_TIME;
      lfb_F_TRIG_Set_Pos : F_TRIG;
   END_VAR
BEGIN
   IF #lx_Init THEN

       // Restart after set Positioning
       IF "gtyp_Setup".x_Set_Pos_Activ OR "gtyp_SSC".x_Start_Park_Position THEN
           #li_StepCase := 0;
       END_IF;

       // falling edge Set Pos
       #lfb_F_TRIG_Set_Pos(CLK := "gtyp_Setup".x_Set_Pos_Activ);

       IF #lfb_F_TRIG_Set_Pos.Q THEN
           #lx_FirstCentre := TRUE;
       END_IF;

       #lfb_TON_Wait(IN := #lx_Start_TON_Wait,
                     PT := #lt_TON_Wait);

       // wait time state
       #lfb_TON_State(IN := NOT #lx_Start_TON_State,
                      PT := T#2s);

       // state of the ssc cyclically transmitted to the cloud
       IF #lfb_TON_State.Q AND NOT #lx_Start_TON_State THEN
           #lx_Start_TON_State := TRUE;
           #li_Return_LDT := RD_SYS_T(#ldt_MQTT);
           "gtyp_Interface_Dashboard".Subscribe.PosPanTiltUnit.ldt_ts := DT_TO_LDT(#ldt_MQTT);
       END_IF;

       // restart wait time state
       IF NOT #lfb_TON_State.Q AND #lx_Start_TON_State THEN
           #lx_Start_TON_State := FALSE;
       END_IF;

       CASE #li_StepCase OF

           0:  // Init
               #lx_Start_TON_State := FALSE;
               "gtyp_SSC".Horizontal_Axis.x_Start_Positioning := FALSE;
               "gtyp_SSC".Vertical_Axis.x_Start_Positioning := FALSE;

               IF NOT "gtyp_Setup".x_Set_Pos_Activ AND NOT "gtyp_SSC".x_Start_Park_Position THEN
                   #li_StepCase := 10;
               END_IF;

           10: // Deciding which route to take 

               IF ("gtyp_Interface_Dashboard".Publish.PosPanTiltUnit.ldt_ts > #lldt_ts_old) OR #lx_FirstCentre THEN

                   #lldt_ts_old := "gtyp_Interface_Dashboard".Publish.PosPanTiltUnit.ldt_ts;

                   // convert the degrees to position
                   #ldi_StepHorizontal := REAL_TO_DINT("FC_Scale_linear"(inr_Y1 := DINT_TO_REAL("gtyp_SSC".Horizontal_Axis.Config.di_Neg_Soft_Switch),
                                                                                                             inr_Y2 := DINT_TO_REAL("gtyp_SSC".Horizontal_Axis.Config.di_Pos_Soft_Switch),
                                                                                                             inr_X1 := 0.0,
                                                                                                             inr_X2 := 180.0,
                                                                                                             inr_X := DINT_TO_REAL("gtyp_Interface_Dashboard".Publish.PosPanTiltUnit.i_degree)));
                   #ldi_StepVertical := REAL_TO_DINT("FC_Scale_linear"(inr_Y1 := DINT_TO_REAL("gtyp_SSC".Vertical_Axis.Config.di_Neg_Soft_Switch),
                                                                                                         inr_Y2 := DINT_TO_REAL("gtyp_SSC".Vertical_Axis.Config.di_Pos_Soft_Switch),
                                                                                                         inr_X1 := 0.0,
                                                                                                         inr_X2 := 180.0,
                                                                                                         inr_X := DINT_TO_REAL("gtyp_Interface_Dashboard".Publish.PosPanTiltUnit.i_degree)));

                   // Procedure - first 
                   IF #lx_FirstCentre THEN
                   #li_StepCase := 20;
                   // Procedure - relmove_left
                   ELSIF ("gtyp_Interface_Dashboard".Publish.PosPanTiltUnit.s_cmd = 'relmove_left')
                       AND (("gtyp_SSC".Horizontal_Axis.di_Actual_Position - #ldi_StepHorizontal) > "gtyp_SSC".Horizontal_Axis.Config.di_Neg_Soft_Switch + 15)
                       AND NOT "IX_SSC_RefSwitchHorizontalAxis_I2" THEN
                       #ldi_TargetPosition_Horizontal := "gtyp_SSC".Horizontal_Axis.di_Actual_Position - #ldi_StepHorizontal;
                       "gtyp_SSC".Horizontal_Axis.di_Target_Position := #ldi_TargetPosition_Horizontal;
                       "gtyp_SSC".Horizontal_Axis.x_Start_Positioning := TRUE;
                       #li_StepCase := 70;
                       // Procedure - relmove_right
                   ELSIF ("gtyp_Interface_Dashboard".Publish.PosPanTiltUnit.s_cmd = 'relmove_right')
                       AND (("gtyp_SSC".Horizontal_Axis.di_Actual_Position + #ldi_StepHorizontal) < "gtyp_SSC".Horizontal_Axis.Config.di_Pos_Soft_Switch - 15) THEN
                       #ldi_TargetPosition_Horizontal := "gtyp_SSC".Horizontal_Axis.di_Actual_Position + #ldi_StepHorizontal;
                       "gtyp_SSC".Horizontal_Axis.di_Target_Position := #ldi_TargetPosition_Horizontal;
                       "gtyp_SSC".Horizontal_Axis.x_Start_Positioning := TRUE;
                       #li_StepCase := 70;
                       // Procedure - relmove_up
                   ELSIF ("gtyp_Interface_Dashboard".Publish.PosPanTiltUnit.s_cmd = 'relmove_up')
                       AND (("gtyp_SSC".Vertical_Axis.di_Actual_Position + #ldi_StepHorizontal) < "gtyp_SSC".Vertical_Axis.Config.di_Pos_Soft_Switch - 15) THEN
                       #ldi_TargetPosition_Vertical := "gtyp_SSC".Vertical_Axis.di_Actual_Position + #ldi_StepVertical;
                       "gtyp_SSC".Vertical_Axis.di_Target_Position := #ldi_TargetPosition_Vertical;
                       "gtyp_SSC".Vertical_Axis.x_Start_Positioning := TRUE;
                       #li_StepCase := 80;
                       // Procedure - relmove_down
                   ELSIF ("gtyp_Interface_Dashboard".Publish.PosPanTiltUnit.s_cmd = 'relmove_down')
                       AND (("gtyp_SSC".Vertical_Axis.di_Actual_Position - #ldi_StepVertical) > "gtyp_SSC".Vertical_Axis.Config.di_Neg_Soft_Switch + 15)
                       AND NOT "IX_SSC_RefSwitchVerticalAxis_I1" THEN
                       #ldi_TargetPosition_Vertical := "gtyp_SSC".Vertical_Axis.di_Actual_Position - #ldi_StepVertical;
                       "gtyp_SSC".Vertical_Axis.di_Target_Position := #ldi_TargetPosition_Vertical;
                       "gtyp_SSC".Vertical_Axis.x_Start_Positioning := TRUE;
                       #li_StepCase := 80;
                       // Procedure - home
                   ELSIF ("gtyp_Interface_Dashboard".Publish.PosPanTiltUnit.s_cmd = 'home') THEN
                       #li_StepCase := 60;
                       // Procedure - start_pan
                   ELSIF ("gtyp_Interface_Dashboard".Publish.PosPanTiltUnit.s_cmd = 'start_pan')
                       AND ("gtyp_SSC".Horizontal_Axis.di_Actual_Position > "gtyp_SSC".Horizontal_Axis.Config.di_Neg_Soft_Switch + 15)
                       AND NOT "IX_SSC_RefSwitchHorizontalAxis_I2" THEN
                       #ldi_TargetPosition_Horizontal := "gtyp_SSC".Horizontal_Axis.Config.di_Neg_Soft_Switch + 15;
                       "gtyp_SSC".Horizontal_Axis.di_Target_Position := #ldi_TargetPosition_Horizontal;
                       "gtyp_SSC".Horizontal_Axis.x_Start_Positioning := TRUE;
                       #li_StepCase := 70;
                       // Procedure - end_pan
                   ELSIF ("gtyp_Interface_Dashboard".Publish.PosPanTiltUnit.s_cmd = 'end_pan')
                       AND ("gtyp_SSC".Horizontal_Axis.di_Actual_Position < "gtyp_SSC".Horizontal_Axis.Config.di_Pos_Soft_Switch - 15) THEN
                       #ldi_TargetPosition_Horizontal := "gtyp_SSC".Horizontal_Axis.Config.di_Pos_Soft_Switch - 15;
                       "gtyp_SSC".Horizontal_Axis.di_Target_Position := #ldi_TargetPosition_Horizontal;
                       "gtyp_SSC".Horizontal_Axis.x_Start_Positioning := TRUE;
                       #li_StepCase := 70;
                       // Procedure - start_tilt
                   ELSIF ("gtyp_Interface_Dashboard".Publish.PosPanTiltUnit.s_cmd = 'start_tilt')
                       AND ("gtyp_SSC".Vertical_Axis.di_Actual_Position > "gtyp_SSC".Vertical_Axis.Config.di_Neg_Soft_Switch + 15)
                       AND NOT "IX_SSC_RefSwitchVerticalAxis_I1" THEN
                       #ldi_TargetPosition_Vertical := "gtyp_SSC".Vertical_Axis.Config.di_Neg_Soft_Switch + 15;
                       "gtyp_SSC".Vertical_Axis.di_Target_Position := #ldi_TargetPosition_Vertical;
                       "gtyp_SSC".Vertical_Axis.x_Start_Positioning := TRUE;
                       #li_StepCase := 80;
                       // Procedure - end_tilt
                   ELSIF ("gtyp_Interface_Dashboard".Publish.PosPanTiltUnit.s_cmd = 'end_tilt')
                       AND ("gtyp_SSC".Vertical_Axis.di_Actual_Position < "gtyp_SSC".Vertical_Axis.Config.di_Pos_Soft_Switch - 15) THEN
                       #ldi_TargetPosition_Vertical := "gtyp_SSC".Vertical_Axis.Config.di_Pos_Soft_Switch - 15;
                       "gtyp_SSC".Vertical_Axis.di_Target_Position := #ldi_TargetPosition_Vertical;
                       "gtyp_SSC".Vertical_Axis.x_Start_Positioning := TRUE;
                       #li_StepCase := 80;
                   END_IF;
               END_IF;

           20: // homing vertical/horizontal axis
               "gtyp_SSC".Horizontal_Axis.x_Reference := TRUE;
               "gtyp_SSC".Vertical_Axis.x_Reference := TRUE;

               IF NOT "gtyp_SSC".Horizontal_Axis.x_Referenced AND NOT "gtyp_SSC".Vertical_Axis.x_Referenced THEN
                   #li_StepCase := 30;
               END_IF;

           30: // homed vertical/horizontal axis
               IF "gtyp_SSC".Horizontal_Axis.x_Referenced THEN
                   "gtyp_SSC".Horizontal_Axis.x_Reference := FALSE;
               END_IF;
               IF "gtyp_SSC".Vertical_Axis.x_Referenced THEN
                   "gtyp_SSC".Vertical_Axis.x_Reference := FALSE;
               END_IF;

               IF "gtyp_SSC".Horizontal_Axis.x_Referenced AND "gtyp_SSC".Vertical_Axis.x_Referenced THEN
                   "gtyp_SSC".Horizontal_Axis.x_Reference := FALSE;
                   "gtyp_SSC".Vertical_Axis.x_Reference := FALSE;
                   #lx_Start_TON_Wait := TRUE;
                   #li_StepCase := 40;
               END_IF;

           40: // wait sequence
               IF #lfb_TON_Wait.Q THEN
                   #lx_Start_TON_Wait := FALSE;
                   #li_StepCase := 50;
               END_IF;

           50: // Position horizontal/vertical axis and reached
               "gtyp_SSC".Horizontal_Axis.di_Target_Position := "gtyp_SSC".di_Pos_HBW_Horizontal;
               "gtyp_SSC".Horizontal_Axis.x_Start_Positioning := TRUE;
               "gtyp_SSC".Vertical_Axis.di_Target_Position := "gtyp_SSC".di_Pos_HBW_Vertical;
               "gtyp_SSC".Vertical_Axis.x_Start_Positioning := TRUE;

               IF ("gtyp_SSC".Horizontal_Axis.di_Actual_Position <= ("gtyp_SSC".di_Pos_HBW_Horizontal + "gtyp_SSC".Horizontal_Axis.Config.di_Pos_Window))
                   AND ("gtyp_SSC".Horizontal_Axis.di_Actual_Position >= ("gtyp_SSC".di_Pos_HBW_Horizontal - "gtyp_SSC".Horizontal_Axis.Config.di_Pos_Window))
                   AND "gtyp_SSC".Horizontal_Axis.x_Position_Reached THEN
                   "gtyp_SSC".Horizontal_Axis.x_Start_Positioning := FALSE;
               END_IF;

               IF ("gtyp_SSC".Vertical_Axis.di_Actual_Position <= ("gtyp_SSC".di_Pos_HBW_Vertical + "gtyp_SSC".Vertical_Axis.Config.di_Pos_Window))
                   AND ("gtyp_SSC".Vertical_Axis.di_Actual_Position >= ("gtyp_SSC".di_Pos_HBW_Vertical - "gtyp_SSC".Vertical_Axis.Config.di_Pos_Window))
                   AND "gtyp_SSC".Vertical_Axis.x_Position_Reached THEN
                   "gtyp_SSC".Vertical_Axis.x_Start_Positioning := FALSE;
               END_IF;

